// TIA Portal V20 export
FUNCTION_BLOCK "LER_Vision_XGX2000_Conversion"   // FB157, LAD
// stored: Access Published, MemoryReserve 100, SetENOAutomatically false
   VAR_INPUT
      VisionData : "LER_typeVisionMonitoring";
   END_VAR
   VAR_OUTPUT
      VisionDataConvert : "LER_typeVisionResultData";
   END_VAR
BEGIN

REGION Network 1: Stack_Width_Judgement Result (0:NONE,1:OK,2:NG)
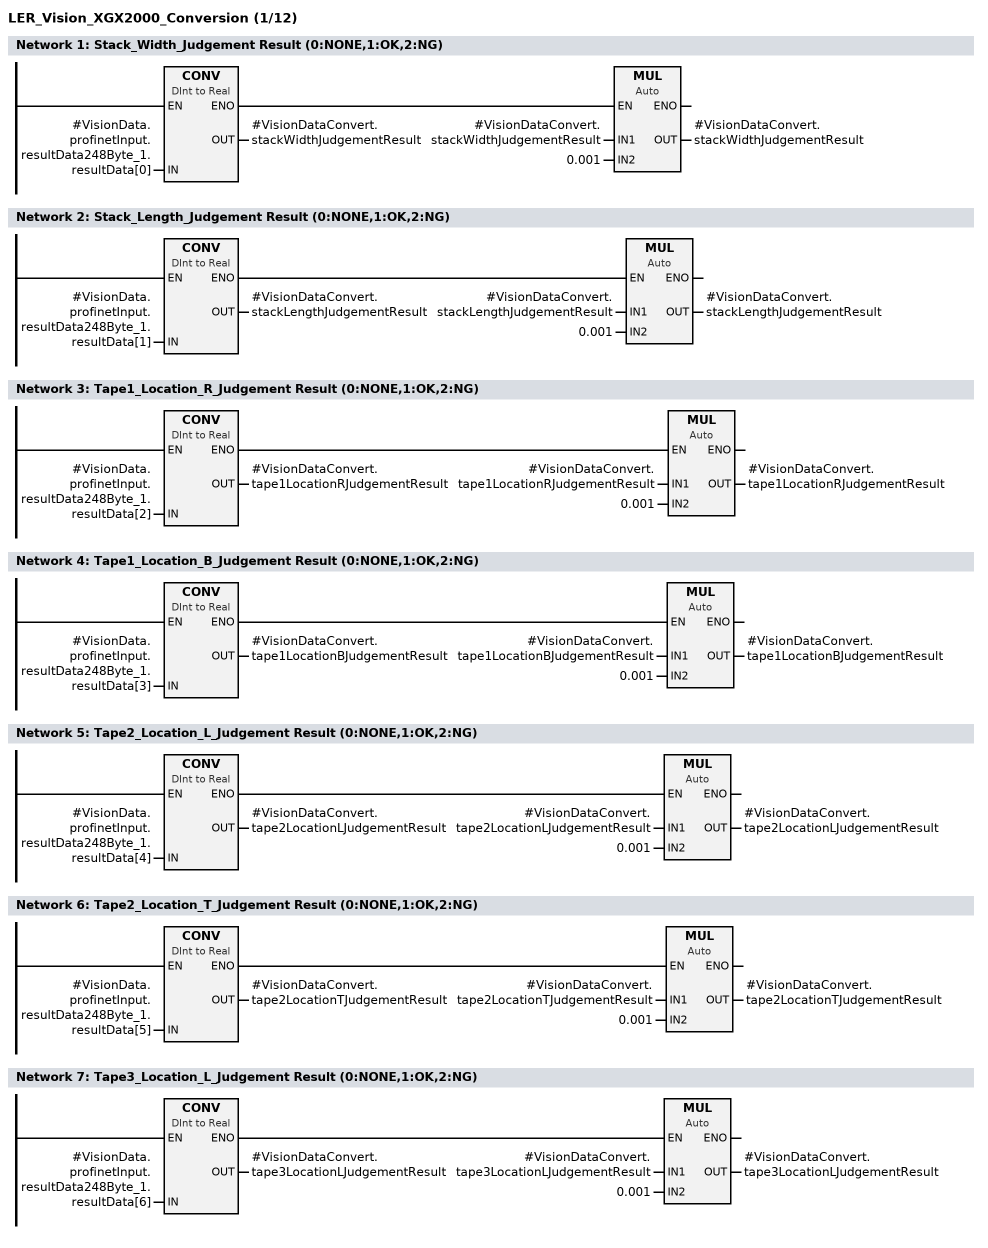
   RUNG wire#powerrail
      { S7_Templates := "[SrcType := DInt, DestType := Real]" } Convert(in := #VisionData.profinetInput.resultData248Byte_1.resultData[0], out => #VisionDataConvert.stackWidthJudgementResult)
      Mul(in1 := #VisionDataConvert.stackWidthJudgementResult, in2 := 0.001, out => #VisionDataConvert.stackWidthJudgementResult)
   END_RUNG
   // the same network as SCL:
   #VisionDataConvert.stackWidthJudgementResult := DINT_TO_REAL(#VisionData.profinetInput.resultData248Byte_1.resultData[0]);
   #VisionDataConvert.stackWidthJudgementResult := #VisionDataConvert.stackWidthJudgementResult * 0.001;
END_REGION

REGION Network 2: Stack_Length_Judgement Result (0:NONE,1:OK,2:NG)
   RUNG wire#powerrail
      { S7_Templates := "[SrcType := DInt, DestType := Real]" } Convert(in := #VisionData.profinetInput.resultData248Byte_1.resultData[1], out => #VisionDataConvert.stackLengthJudgementResult)
      Mul(in1 := #VisionDataConvert.stackLengthJudgementResult, in2 := 0.001, out => #VisionDataConvert.stackLengthJudgementResult)
   END_RUNG
   // the same network as SCL:
   #VisionDataConvert.stackLengthJudgementResult := DINT_TO_REAL(#VisionData.profinetInput.resultData248Byte_1.resultData[1]);
   #VisionDataConvert.stackLengthJudgementResult := #VisionDataConvert.stackLengthJudgementResult * 0.001;
END_REGION

REGION Network 3: Tape1_Location_R_Judgement Result (0:NONE,1:OK,2:NG)
   RUNG wire#powerrail
      { S7_Templates := "[SrcType := DInt, DestType := Real]" } Convert(in := #VisionData.profinetInput.resultData248Byte_1.resultData[2], out => #VisionDataConvert.tape1LocationRJudgementResult)
      Mul(in1 := #VisionDataConvert.tape1LocationRJudgementResult, in2 := 0.001, out => #VisionDataConvert.tape1LocationRJudgementResult)
   END_RUNG
   // the same network as SCL:
   #VisionDataConvert.tape1LocationRJudgementResult := DINT_TO_REAL(#VisionData.profinetInput.resultData248Byte_1.resultData[2]);
   #VisionDataConvert.tape1LocationRJudgementResult := #VisionDataConvert.tape1LocationRJudgementResult * 0.001;
END_REGION

REGION Network 4: Tape1_Location_B_Judgement Result (0:NONE,1:OK,2:NG)
   RUNG wire#powerrail
      { S7_Templates := "[SrcType := DInt, DestType := Real]" } Convert(in := #VisionData.profinetInput.resultData248Byte_1.resultData[3], out => #VisionDataConvert.tape1LocationBJudgementResult)
      Mul(in1 := #VisionDataConvert.tape1LocationBJudgementResult, in2 := 0.001, out => #VisionDataConvert.tape1LocationBJudgementResult)
   END_RUNG
   // the same network as SCL:
   #VisionDataConvert.tape1LocationBJudgementResult := DINT_TO_REAL(#VisionData.profinetInput.resultData248Byte_1.resultData[3]);
   #VisionDataConvert.tape1LocationBJudgementResult := #VisionDataConvert.tape1LocationBJudgementResult * 0.001;
END_REGION

REGION Network 5: Tape2_Location_L_Judgement Result (0:NONE,1:OK,2:NG)
   RUNG wire#powerrail
      { S7_Templates := "[SrcType := DInt, DestType := Real]" } Convert(in := #VisionData.profinetInput.resultData248Byte_1.resultData[4], out => #VisionDataConvert.tape2LocationLJudgementResult)
      Mul(in1 := #VisionDataConvert.tape2LocationLJudgementResult, in2 := 0.001, out => #VisionDataConvert.tape2LocationLJudgementResult)
   END_RUNG
   // the same network as SCL:
   #VisionDataConvert.tape2LocationLJudgementResult := DINT_TO_REAL(#VisionData.profinetInput.resultData248Byte_1.resultData[4]);
   #VisionDataConvert.tape2LocationLJudgementResult := #VisionDataConvert.tape2LocationLJudgementResult * 0.001;
END_REGION

REGION Network 6: Tape2_Location_T_Judgement Result (0:NONE,1:OK,2:NG)
   RUNG wire#powerrail
      { S7_Templates := "[SrcType := DInt, DestType := Real]" } Convert(in := #VisionData.profinetInput.resultData248Byte_1.resultData[5], out => #VisionDataConvert.tape2LocationTJudgementResult)
      Mul(in1 := #VisionDataConvert.tape2LocationTJudgementResult, in2 := 0.001, out => #VisionDataConvert.tape2LocationTJudgementResult)
   END_RUNG
   // the same network as SCL:
   #VisionDataConvert.tape2LocationTJudgementResult := DINT_TO_REAL(#VisionData.profinetInput.resultData248Byte_1.resultData[5]);
   #VisionDataConvert.tape2LocationTJudgementResult := #VisionDataConvert.tape2LocationTJudgementResult * 0.001;
END_REGION

REGION Network 7: Tape3_Location_L_Judgement Result (0:NONE,1:OK,2:NG)
   RUNG wire#powerrail
      { S7_Templates := "[SrcType := DInt, DestType := Real]" } Convert(in := #VisionData.profinetInput.resultData248Byte_1.resultData[6], out => #VisionDataConvert.tape3LocationLJudgementResult)
      Mul(in1 := #VisionDataConvert.tape3LocationLJudgementResult, in2 := 0.001, out => #VisionDataConvert.tape3LocationLJudgementResult)
   END_RUNG
   // the same network as SCL:
   #VisionDataConvert.tape3LocationLJudgementResult := DINT_TO_REAL(#VisionData.profinetInput.resultData248Byte_1.resultData[6]);
   #VisionDataConvert.tape3LocationLJudgementResult := #VisionDataConvert.tape3LocationLJudgementResult * 0.001;
END_REGION

REGION Network 8: Tape3_Location_B_Judgement Result (0:NONE,1:OK,2:NG)
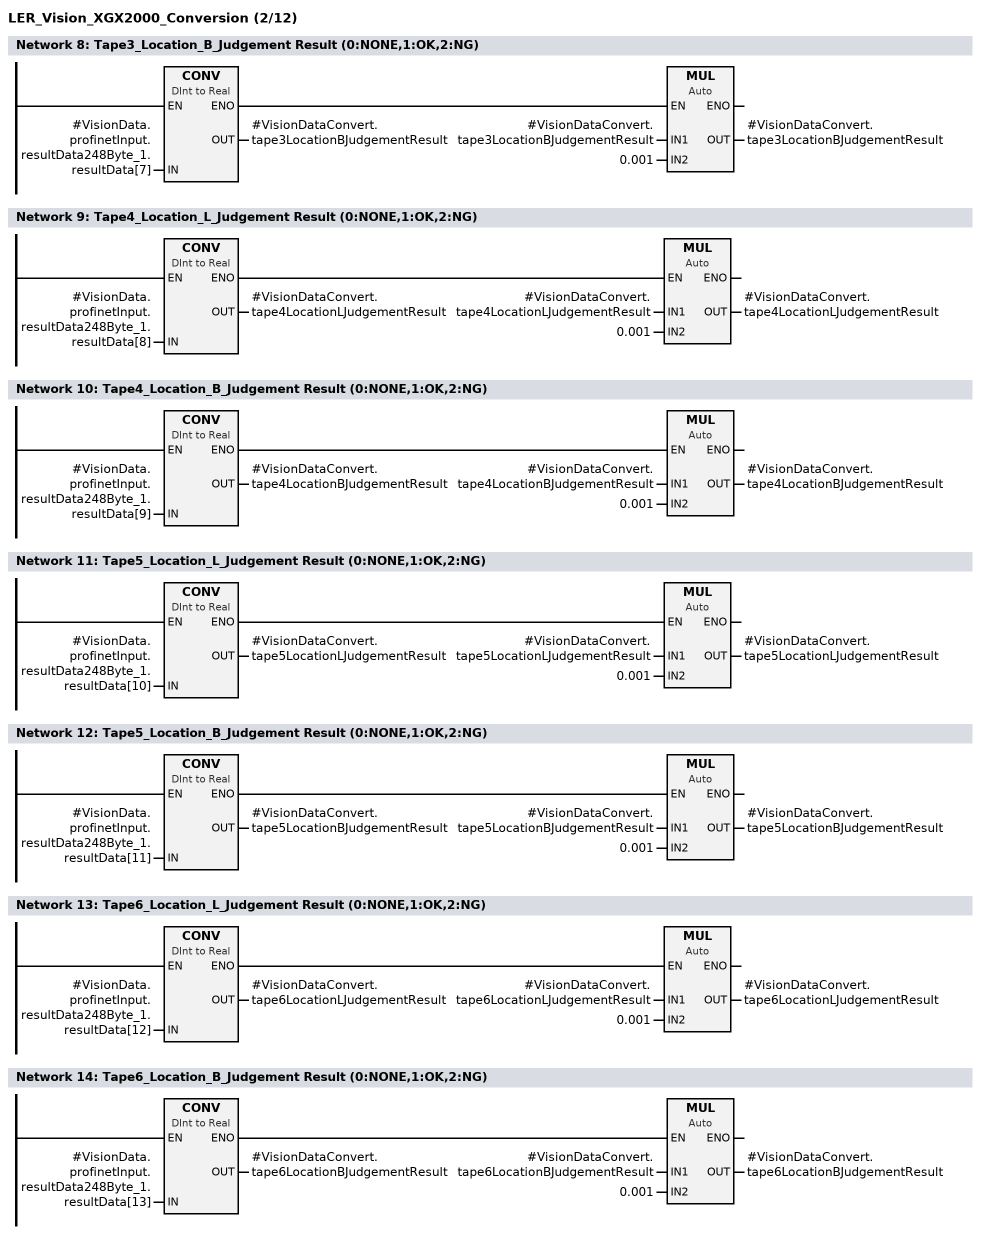
   RUNG wire#powerrail
      { S7_Templates := "[SrcType := DInt, DestType := Real]" } Convert(in := #VisionData.profinetInput.resultData248Byte_1.resultData[7], out => #VisionDataConvert.tape3LocationBJudgementResult)
      Mul(in1 := #VisionDataConvert.tape3LocationBJudgementResult, in2 := 0.001, out => #VisionDataConvert.tape3LocationBJudgementResult)
   END_RUNG
   // the same network as SCL:
   #VisionDataConvert.tape3LocationBJudgementResult := DINT_TO_REAL(#VisionData.profinetInput.resultData248Byte_1.resultData[7]);
   #VisionDataConvert.tape3LocationBJudgementResult := #VisionDataConvert.tape3LocationBJudgementResult * 0.001;
END_REGION

REGION Network 9: Tape4_Location_L_Judgement Result (0:NONE,1:OK,2:NG)
   RUNG wire#powerrail
      { S7_Templates := "[SrcType := DInt, DestType := Real]" } Convert(in := #VisionData.profinetInput.resultData248Byte_1.resultData[8], out => #VisionDataConvert.tape4LocationLJudgementResult)
      Mul(in1 := #VisionDataConvert.tape4LocationLJudgementResult, in2 := 0.001, out => #VisionDataConvert.tape4LocationLJudgementResult)
   END_RUNG
   // the same network as SCL:
   #VisionDataConvert.tape4LocationLJudgementResult := DINT_TO_REAL(#VisionData.profinetInput.resultData248Byte_1.resultData[8]);
   #VisionDataConvert.tape4LocationLJudgementResult := #VisionDataConvert.tape4LocationLJudgementResult * 0.001;
END_REGION

REGION Network 10: Tape4_Location_B_Judgement Result (0:NONE,1:OK,2:NG)
   RUNG wire#powerrail
      { S7_Templates := "[SrcType := DInt, DestType := Real]" } Convert(in := #VisionData.profinetInput.resultData248Byte_1.resultData[9], out => #VisionDataConvert.tape4LocationBJudgementResult)
      Mul(in1 := #VisionDataConvert.tape4LocationBJudgementResult, in2 := 0.001, out => #VisionDataConvert.tape4LocationBJudgementResult)
   END_RUNG
   // the same network as SCL:
   #VisionDataConvert.tape4LocationBJudgementResult := DINT_TO_REAL(#VisionData.profinetInput.resultData248Byte_1.resultData[9]);
   #VisionDataConvert.tape4LocationBJudgementResult := #VisionDataConvert.tape4LocationBJudgementResult * 0.001;
END_REGION

REGION Network 11: Tape5_Location_L_Judgement Result (0:NONE,1:OK,2:NG)
   RUNG wire#powerrail
      { S7_Templates := "[SrcType := DInt, DestType := Real]" } Convert(in := #VisionData.profinetInput.resultData248Byte_1.resultData[10], out => #VisionDataConvert.tape5LocationLJudgementResult)
      Mul(in1 := #VisionDataConvert.tape5LocationLJudgementResult, in2 := 0.001, out => #VisionDataConvert.tape5LocationLJudgementResult)
   END_RUNG
   // the same network as SCL:
   #VisionDataConvert.tape5LocationLJudgementResult := DINT_TO_REAL(#VisionData.profinetInput.resultData248Byte_1.resultData[10]);
   #VisionDataConvert.tape5LocationLJudgementResult := #VisionDataConvert.tape5LocationLJudgementResult * 0.001;
END_REGION

REGION Network 12: Tape5_Location_B_Judgement Result (0:NONE,1:OK,2:NG)
   RUNG wire#powerrail
      { S7_Templates := "[SrcType := DInt, DestType := Real]" } Convert(in := #VisionData.profinetInput.resultData248Byte_1.resultData[11], out => #VisionDataConvert.tape5LocationBJudgementResult)
      Mul(in1 := #VisionDataConvert.tape5LocationBJudgementResult, in2 := 0.001, out => #VisionDataConvert.tape5LocationBJudgementResult)
   END_RUNG
   // the same network as SCL:
   #VisionDataConvert.tape5LocationBJudgementResult := DINT_TO_REAL(#VisionData.profinetInput.resultData248Byte_1.resultData[11]);
   #VisionDataConvert.tape5LocationBJudgementResult := #VisionDataConvert.tape5LocationBJudgementResult * 0.001;
END_REGION

REGION Network 13: Tape6_Location_L_Judgement Result (0:NONE,1:OK,2:NG)
   RUNG wire#powerrail
      { S7_Templates := "[SrcType := DInt, DestType := Real]" } Convert(in := #VisionData.profinetInput.resultData248Byte_1.resultData[12], out => #VisionDataConvert.tape6LocationLJudgementResult)
      Mul(in1 := #VisionDataConvert.tape6LocationLJudgementResult, in2 := 0.001, out => #VisionDataConvert.tape6LocationLJudgementResult)
   END_RUNG
   // the same network as SCL:
   #VisionDataConvert.tape6LocationLJudgementResult := DINT_TO_REAL(#VisionData.profinetInput.resultData248Byte_1.resultData[12]);
   #VisionDataConvert.tape6LocationLJudgementResult := #VisionDataConvert.tape6LocationLJudgementResult * 0.001;
END_REGION

REGION Network 14: Tape6_Location_B_Judgement Result (0:NONE,1:OK,2:NG)
   RUNG wire#powerrail
      { S7_Templates := "[SrcType := DInt, DestType := Real]" } Convert(in := #VisionData.profinetInput.resultData248Byte_1.resultData[13], out => #VisionDataConvert.tape6LocationBJudgementResult)
      Mul(in1 := #VisionDataConvert.tape6LocationBJudgementResult, in2 := 0.001, out => #VisionDataConvert.tape6LocationBJudgementResult)
   END_RUNG
   // the same network as SCL:
   #VisionDataConvert.tape6LocationBJudgementResult := DINT_TO_REAL(#VisionData.profinetInput.resultData248Byte_1.resultData[13]);
   #VisionDataConvert.tape6LocationBJudgementResult := #VisionDataConvert.tape6LocationBJudgementResult * 0.001;
END_REGION

REGION Network 15: Tape7_Location_L_Judgement Result (0:NONE,1:OK,2:NG)
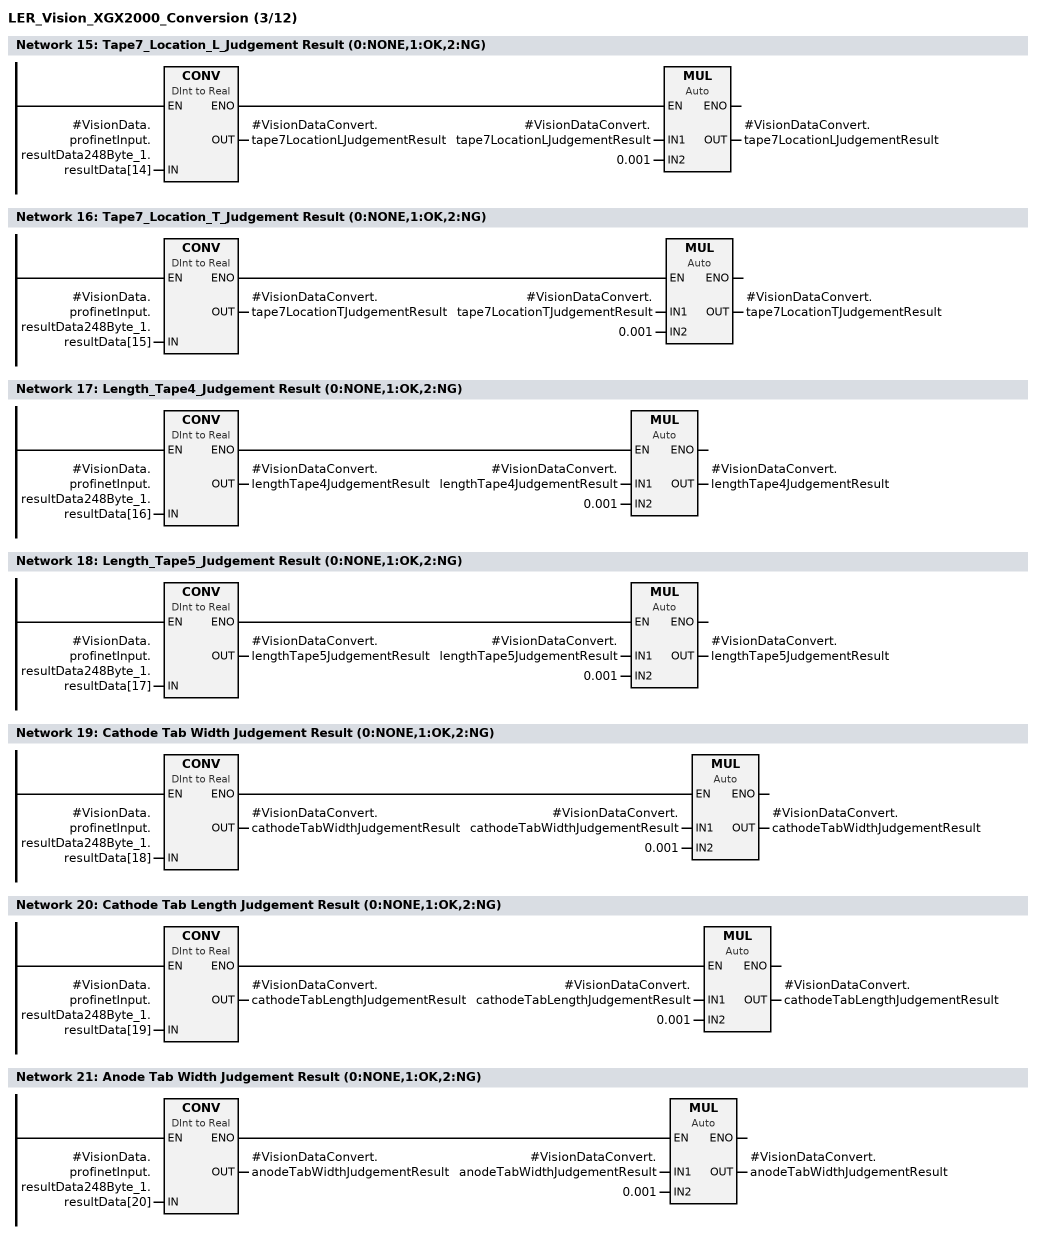
   RUNG wire#powerrail
      { S7_Templates := "[SrcType := DInt, DestType := Real]" } Convert(in := #VisionData.profinetInput.resultData248Byte_1.resultData[14], out => #VisionDataConvert.tape7LocationLJudgementResult)
      Mul(in1 := #VisionDataConvert.tape7LocationLJudgementResult, in2 := 0.001, out => #VisionDataConvert.tape7LocationLJudgementResult)
   END_RUNG
   // the same network as SCL:
   #VisionDataConvert.tape7LocationLJudgementResult := DINT_TO_REAL(#VisionData.profinetInput.resultData248Byte_1.resultData[14]);
   #VisionDataConvert.tape7LocationLJudgementResult := #VisionDataConvert.tape7LocationLJudgementResult * 0.001;
END_REGION

REGION Network 16: Tape7_Location_T_Judgement Result (0:NONE,1:OK,2:NG)
   RUNG wire#powerrail
      { S7_Templates := "[SrcType := DInt, DestType := Real]" } Convert(in := #VisionData.profinetInput.resultData248Byte_1.resultData[15], out => #VisionDataConvert.tape7LocationTJudgementResult)
      Mul(in1 := #VisionDataConvert.tape7LocationTJudgementResult, in2 := 0.001, out => #VisionDataConvert.tape7LocationTJudgementResult)
   END_RUNG
   // the same network as SCL:
   #VisionDataConvert.tape7LocationTJudgementResult := DINT_TO_REAL(#VisionData.profinetInput.resultData248Byte_1.resultData[15]);
   #VisionDataConvert.tape7LocationTJudgementResult := #VisionDataConvert.tape7LocationTJudgementResult * 0.001;
END_REGION

REGION Network 17: Length_Tape4_Judgement Result (0:NONE,1:OK,2:NG)
   RUNG wire#powerrail
      { S7_Templates := "[SrcType := DInt, DestType := Real]" } Convert(in := #VisionData.profinetInput.resultData248Byte_1.resultData[16], out => #VisionDataConvert.lengthTape4JudgementResult)
      Mul(in1 := #VisionDataConvert.lengthTape4JudgementResult, in2 := 0.001, out => #VisionDataConvert.lengthTape4JudgementResult)
   END_RUNG
   // the same network as SCL:
   #VisionDataConvert.lengthTape4JudgementResult := DINT_TO_REAL(#VisionData.profinetInput.resultData248Byte_1.resultData[16]);
   #VisionDataConvert.lengthTape4JudgementResult := #VisionDataConvert.lengthTape4JudgementResult * 0.001;
END_REGION

REGION Network 18: Length_Tape5_Judgement Result (0:NONE,1:OK,2:NG)
   RUNG wire#powerrail
      { S7_Templates := "[SrcType := DInt, DestType := Real]" } Convert(in := #VisionData.profinetInput.resultData248Byte_1.resultData[17], out => #VisionDataConvert.lengthTape5JudgementResult)
      Mul(in1 := #VisionDataConvert.lengthTape5JudgementResult, in2 := 0.001, out => #VisionDataConvert.lengthTape5JudgementResult)
   END_RUNG
   // the same network as SCL:
   #VisionDataConvert.lengthTape5JudgementResult := DINT_TO_REAL(#VisionData.profinetInput.resultData248Byte_1.resultData[17]);
   #VisionDataConvert.lengthTape5JudgementResult := #VisionDataConvert.lengthTape5JudgementResult * 0.001;
END_REGION

REGION Network 19: Cathode Tab Width Judgement Result (0:NONE,1:OK,2:NG)
   RUNG wire#powerrail
      { S7_Templates := "[SrcType := DInt, DestType := Real]" } Convert(in := #VisionData.profinetInput.resultData248Byte_1.resultData[18], out => #VisionDataConvert.cathodeTabWidthJudgementResult)
      Mul(in1 := #VisionDataConvert.cathodeTabWidthJudgementResult, in2 := 0.001, out => #VisionDataConvert.cathodeTabWidthJudgementResult)
   END_RUNG
   // the same network as SCL:
   #VisionDataConvert.cathodeTabWidthJudgementResult := DINT_TO_REAL(#VisionData.profinetInput.resultData248Byte_1.resultData[18]);
   #VisionDataConvert.cathodeTabWidthJudgementResult := #VisionDataConvert.cathodeTabWidthJudgementResult * 0.001;
END_REGION

REGION Network 20: Cathode Tab Length Judgement Result (0:NONE,1:OK,2:NG)
   RUNG wire#powerrail
      { S7_Templates := "[SrcType := DInt, DestType := Real]" } Convert(in := #VisionData.profinetInput.resultData248Byte_1.resultData[19], out => #VisionDataConvert.cathodeTabLengthJudgementResult)
      Mul(in1 := #VisionDataConvert.cathodeTabLengthJudgementResult, in2 := 0.001, out => #VisionDataConvert.cathodeTabLengthJudgementResult)
   END_RUNG
   // the same network as SCL:
   #VisionDataConvert.cathodeTabLengthJudgementResult := DINT_TO_REAL(#VisionData.profinetInput.resultData248Byte_1.resultData[19]);
   #VisionDataConvert.cathodeTabLengthJudgementResult := #VisionDataConvert.cathodeTabLengthJudgementResult * 0.001;
END_REGION

REGION Network 21: Anode Tab Width Judgement Result (0:NONE,1:OK,2:NG)
   RUNG wire#powerrail
      { S7_Templates := "[SrcType := DInt, DestType := Real]" } Convert(in := #VisionData.profinetInput.resultData248Byte_1.resultData[20], out => #VisionDataConvert.anodeTabWidthJudgementResult)
      Mul(in1 := #VisionDataConvert.anodeTabWidthJudgementResult, in2 := 0.001, out => #VisionDataConvert.anodeTabWidthJudgementResult)
   END_RUNG
   // the same network as SCL:
   #VisionDataConvert.anodeTabWidthJudgementResult := DINT_TO_REAL(#VisionData.profinetInput.resultData248Byte_1.resultData[20]);
   #VisionDataConvert.anodeTabWidthJudgementResult := #VisionDataConvert.anodeTabWidthJudgementResult * 0.001;
END_REGION

REGION Network 22: Anode Tab Length Judgement Result (0:NONE,1:OK,2:NG)
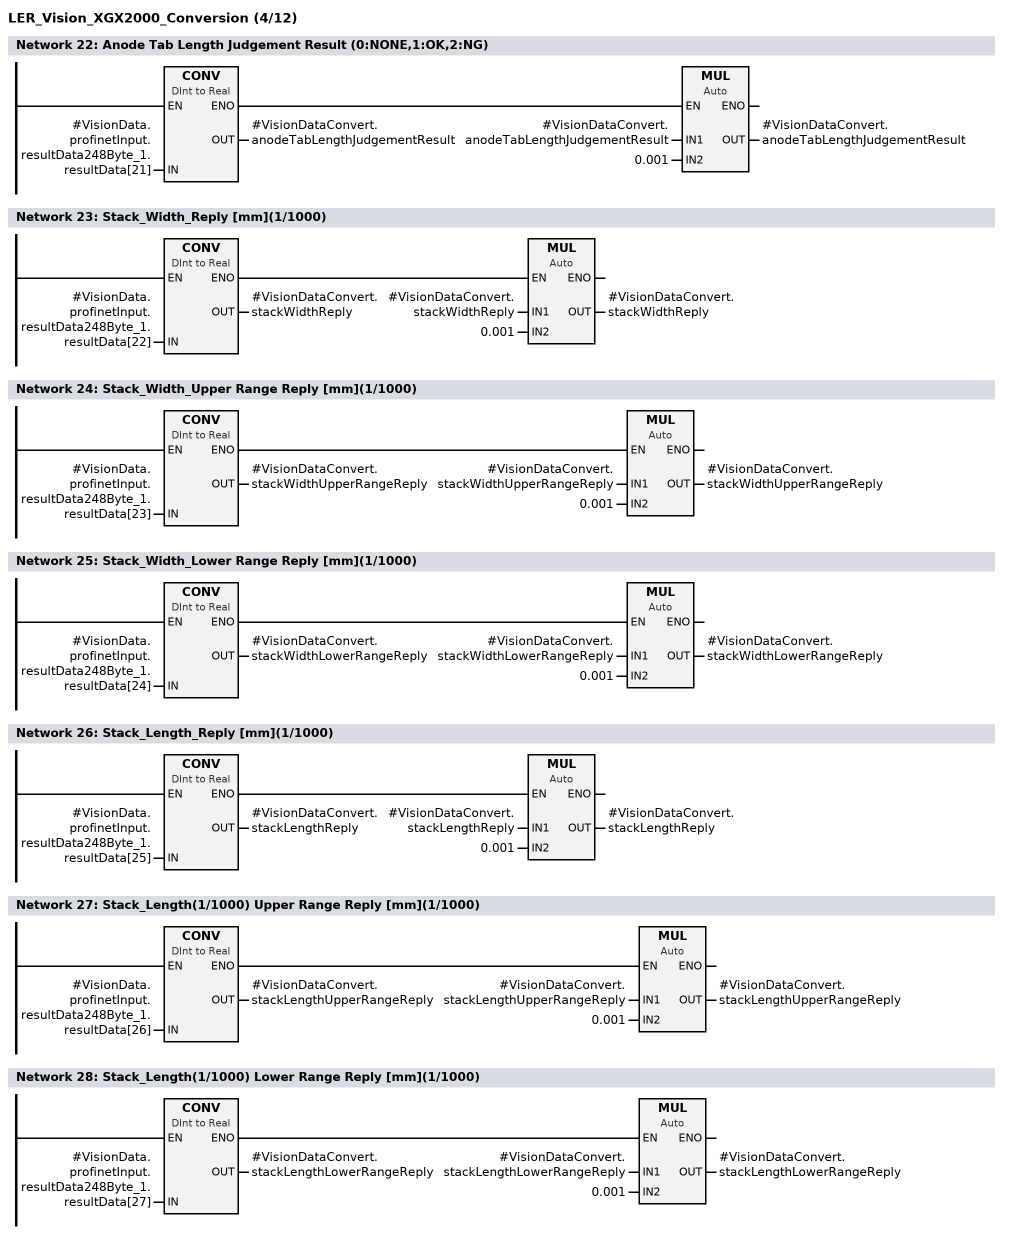
   RUNG wire#powerrail
      { S7_Templates := "[SrcType := DInt, DestType := Real]" } Convert(in := #VisionData.profinetInput.resultData248Byte_1.resultData[21], out => #VisionDataConvert.anodeTabLengthJudgementResult)
      Mul(in1 := #VisionDataConvert.anodeTabLengthJudgementResult, in2 := 0.001, out => #VisionDataConvert.anodeTabLengthJudgementResult)
   END_RUNG
   // the same network as SCL:
   #VisionDataConvert.anodeTabLengthJudgementResult := DINT_TO_REAL(#VisionData.profinetInput.resultData248Byte_1.resultData[21]);
   #VisionDataConvert.anodeTabLengthJudgementResult := #VisionDataConvert.anodeTabLengthJudgementResult * 0.001;
END_REGION

REGION Network 23: Stack_Width_Reply [mm](1/1000)
   RUNG wire#powerrail
      { S7_Templates := "[SrcType := DInt, DestType := Real]" } Convert(in := #VisionData.profinetInput.resultData248Byte_1.resultData[22], out => #VisionDataConvert.stackWidthReply)
      Mul(in1 := #VisionDataConvert.stackWidthReply, in2 := 0.001, out => #VisionDataConvert.stackWidthReply)
   END_RUNG
   // the same network as SCL:
   #VisionDataConvert.stackWidthReply := DINT_TO_REAL(#VisionData.profinetInput.resultData248Byte_1.resultData[22]);
   #VisionDataConvert.stackWidthReply := #VisionDataConvert.stackWidthReply * 0.001;
END_REGION

REGION Network 24: Stack_Width_Upper Range Reply [mm](1/1000)
   RUNG wire#powerrail
      { S7_Templates := "[SrcType := DInt, DestType := Real]" } Convert(in := #VisionData.profinetInput.resultData248Byte_1.resultData[23], out => #VisionDataConvert.stackWidthUpperRangeReply)
      Mul(in1 := #VisionDataConvert.stackWidthUpperRangeReply, in2 := 0.001, out => #VisionDataConvert.stackWidthUpperRangeReply)
   END_RUNG
   // the same network as SCL:
   #VisionDataConvert.stackWidthUpperRangeReply := DINT_TO_REAL(#VisionData.profinetInput.resultData248Byte_1.resultData[23]);
   #VisionDataConvert.stackWidthUpperRangeReply := #VisionDataConvert.stackWidthUpperRangeReply * 0.001;
END_REGION

REGION Network 25: Stack_Width_Lower Range Reply [mm](1/1000)
   RUNG wire#powerrail
      { S7_Templates := "[SrcType := DInt, DestType := Real]" } Convert(in := #VisionData.profinetInput.resultData248Byte_1.resultData[24], out => #VisionDataConvert.stackWidthLowerRangeReply)
      Mul(in1 := #VisionDataConvert.stackWidthLowerRangeReply, in2 := 0.001, out => #VisionDataConvert.stackWidthLowerRangeReply)
   END_RUNG
   // the same network as SCL:
   #VisionDataConvert.stackWidthLowerRangeReply := DINT_TO_REAL(#VisionData.profinetInput.resultData248Byte_1.resultData[24]);
   #VisionDataConvert.stackWidthLowerRangeReply := #VisionDataConvert.stackWidthLowerRangeReply * 0.001;
END_REGION

REGION Network 26: Stack_Length_Reply [mm](1/1000)
   RUNG wire#powerrail
      { S7_Templates := "[SrcType := DInt, DestType := Real]" } Convert(in := #VisionData.profinetInput.resultData248Byte_1.resultData[25], out => #VisionDataConvert.stackLengthReply)
      Mul(in1 := #VisionDataConvert.stackLengthReply, in2 := 0.001, out => #VisionDataConvert.stackLengthReply)
   END_RUNG
   // the same network as SCL:
   #VisionDataConvert.stackLengthReply := DINT_TO_REAL(#VisionData.profinetInput.resultData248Byte_1.resultData[25]);
   #VisionDataConvert.stackLengthReply := #VisionDataConvert.stackLengthReply * 0.001;
END_REGION

REGION Network 27: Stack_Length(1/1000) Upper Range Reply [mm](1/1000)
   RUNG wire#powerrail
      { S7_Templates := "[SrcType := DInt, DestType := Real]" } Convert(in := #VisionData.profinetInput.resultData248Byte_1.resultData[26], out => #VisionDataConvert.stackLengthUpperRangeReply)
      Mul(in1 := #VisionDataConvert.stackLengthUpperRangeReply, in2 := 0.001, out => #VisionDataConvert.stackLengthUpperRangeReply)
   END_RUNG
   // the same network as SCL:
   #VisionDataConvert.stackLengthUpperRangeReply := DINT_TO_REAL(#VisionData.profinetInput.resultData248Byte_1.resultData[26]);
   #VisionDataConvert.stackLengthUpperRangeReply := #VisionDataConvert.stackLengthUpperRangeReply * 0.001;
END_REGION

REGION Network 28: Stack_Length(1/1000) Lower Range Reply [mm](1/1000)
   RUNG wire#powerrail
      { S7_Templates := "[SrcType := DInt, DestType := Real]" } Convert(in := #VisionData.profinetInput.resultData248Byte_1.resultData[27], out => #VisionDataConvert.stackLengthLowerRangeReply)
      Mul(in1 := #VisionDataConvert.stackLengthLowerRangeReply, in2 := 0.001, out => #VisionDataConvert.stackLengthLowerRangeReply)
   END_RUNG
   // the same network as SCL:
   #VisionDataConvert.stackLengthLowerRangeReply := DINT_TO_REAL(#VisionData.profinetInput.resultData248Byte_1.resultData[27]);
   #VisionDataConvert.stackLengthLowerRangeReply := #VisionDataConvert.stackLengthLowerRangeReply * 0.001;
END_REGION

REGION Network 29: Tape1_Location_R_Reply [mm](1/1000)
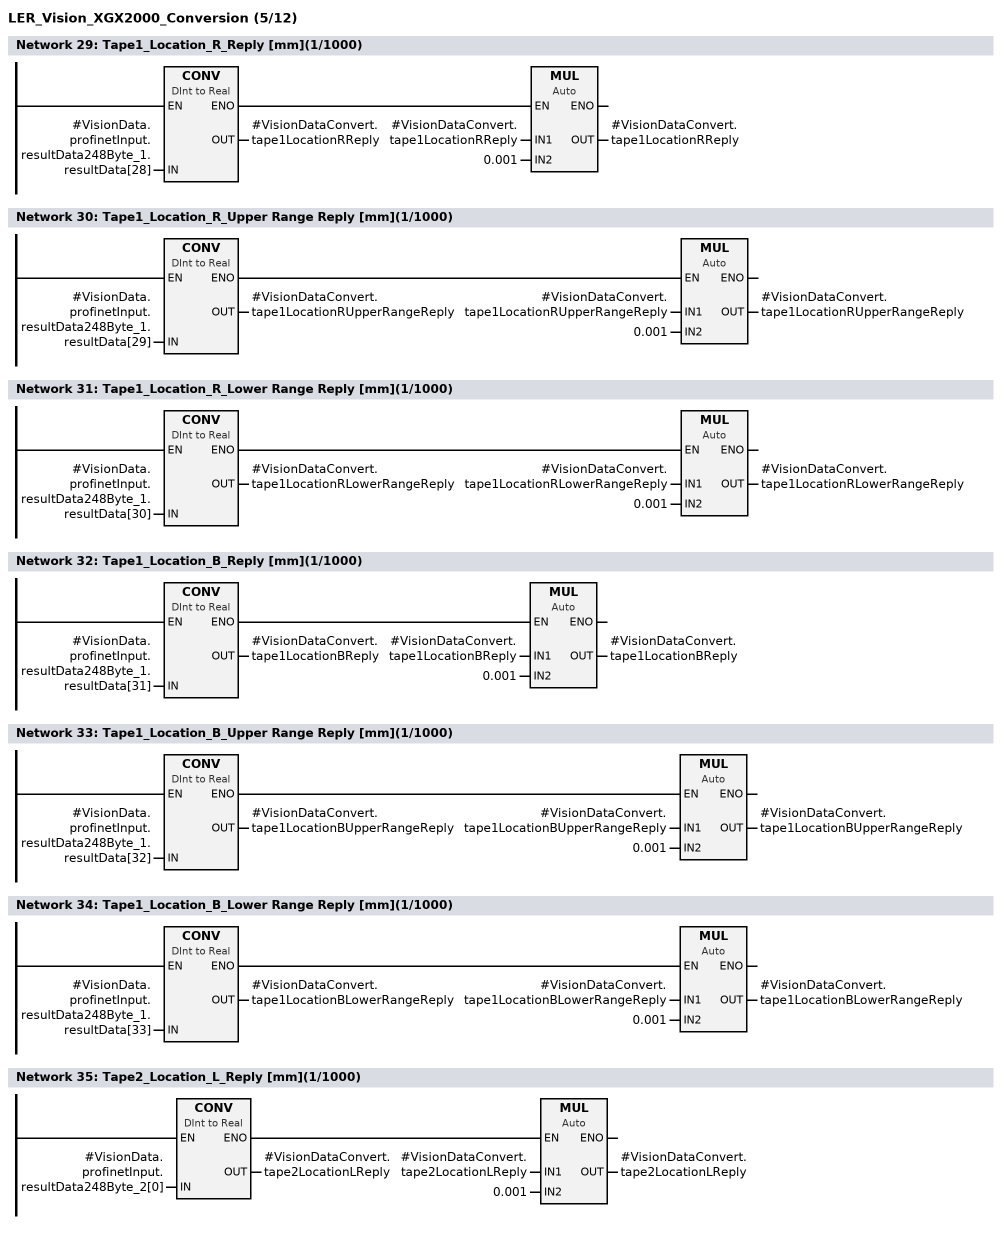
   RUNG wire#powerrail
      { S7_Templates := "[SrcType := DInt, DestType := Real]" } Convert(in := #VisionData.profinetInput.resultData248Byte_1.resultData[28], out => #VisionDataConvert.tape1LocationRReply)
      Mul(in1 := #VisionDataConvert.tape1LocationRReply, in2 := 0.001, out => #VisionDataConvert.tape1LocationRReply)
   END_RUNG
   // the same network as SCL:
   #VisionDataConvert.tape1LocationRReply := DINT_TO_REAL(#VisionData.profinetInput.resultData248Byte_1.resultData[28]);
   #VisionDataConvert.tape1LocationRReply := #VisionDataConvert.tape1LocationRReply * 0.001;
END_REGION

REGION Network 30: Tape1_Location_R_Upper Range Reply [mm](1/1000)
   RUNG wire#powerrail
      { S7_Templates := "[SrcType := DInt, DestType := Real]" } Convert(in := #VisionData.profinetInput.resultData248Byte_1.resultData[29], out => #VisionDataConvert.tape1LocationRUpperRangeReply)
      Mul(in1 := #VisionDataConvert.tape1LocationRUpperRangeReply, in2 := 0.001, out => #VisionDataConvert.tape1LocationRUpperRangeReply)
   END_RUNG
   // the same network as SCL:
   #VisionDataConvert.tape1LocationRUpperRangeReply := DINT_TO_REAL(#VisionData.profinetInput.resultData248Byte_1.resultData[29]);
   #VisionDataConvert.tape1LocationRUpperRangeReply := #VisionDataConvert.tape1LocationRUpperRangeReply * 0.001;
END_REGION

REGION Network 31: Tape1_Location_R_Lower Range Reply [mm](1/1000)
   RUNG wire#powerrail
      { S7_Templates := "[SrcType := DInt, DestType := Real]" } Convert(in := #VisionData.profinetInput.resultData248Byte_1.resultData[30], out => #VisionDataConvert.tape1LocationRLowerRangeReply)
      Mul(in1 := #VisionDataConvert.tape1LocationRLowerRangeReply, in2 := 0.001, out => #VisionDataConvert.tape1LocationRLowerRangeReply)
   END_RUNG
   // the same network as SCL:
   #VisionDataConvert.tape1LocationRLowerRangeReply := DINT_TO_REAL(#VisionData.profinetInput.resultData248Byte_1.resultData[30]);
   #VisionDataConvert.tape1LocationRLowerRangeReply := #VisionDataConvert.tape1LocationRLowerRangeReply * 0.001;
END_REGION

REGION Network 32: Tape1_Location_B_Reply [mm](1/1000)
   RUNG wire#powerrail
      { S7_Templates := "[SrcType := DInt, DestType := Real]" } Convert(in := #VisionData.profinetInput.resultData248Byte_1.resultData[31], out => #VisionDataConvert.tape1LocationBReply)
      Mul(in1 := #VisionDataConvert.tape1LocationBReply, in2 := 0.001, out => #VisionDataConvert.tape1LocationBReply)
   END_RUNG
   // the same network as SCL:
   #VisionDataConvert.tape1LocationBReply := DINT_TO_REAL(#VisionData.profinetInput.resultData248Byte_1.resultData[31]);
   #VisionDataConvert.tape1LocationBReply := #VisionDataConvert.tape1LocationBReply * 0.001;
END_REGION

REGION Network 33: Tape1_Location_B_Upper Range Reply [mm](1/1000)
   RUNG wire#powerrail
      { S7_Templates := "[SrcType := DInt, DestType := Real]" } Convert(in := #VisionData.profinetInput.resultData248Byte_1.resultData[32], out => #VisionDataConvert.tape1LocationBUpperRangeReply)
      Mul(in1 := #VisionDataConvert.tape1LocationBUpperRangeReply, in2 := 0.001, out => #VisionDataConvert.tape1LocationBUpperRangeReply)
   END_RUNG
   // the same network as SCL:
   #VisionDataConvert.tape1LocationBUpperRangeReply := DINT_TO_REAL(#VisionData.profinetInput.resultData248Byte_1.resultData[32]);
   #VisionDataConvert.tape1LocationBUpperRangeReply := #VisionDataConvert.tape1LocationBUpperRangeReply * 0.001;
END_REGION

REGION Network 34: Tape1_Location_B_Lower Range Reply [mm](1/1000)
   RUNG wire#powerrail
      { S7_Templates := "[SrcType := DInt, DestType := Real]" } Convert(in := #VisionData.profinetInput.resultData248Byte_1.resultData[33], out => #VisionDataConvert.tape1LocationBLowerRangeReply)
      Mul(in1 := #VisionDataConvert.tape1LocationBLowerRangeReply, in2 := 0.001, out => #VisionDataConvert.tape1LocationBLowerRangeReply)
   END_RUNG
   // the same network as SCL:
   #VisionDataConvert.tape1LocationBLowerRangeReply := DINT_TO_REAL(#VisionData.profinetInput.resultData248Byte_1.resultData[33]);
   #VisionDataConvert.tape1LocationBLowerRangeReply := #VisionDataConvert.tape1LocationBLowerRangeReply * 0.001;
END_REGION

REGION Network 35: Tape2_Location_L_Reply [mm](1/1000)
   RUNG wire#powerrail
      { S7_Templates := "[SrcType := DInt, DestType := Real]" } Convert(in := #VisionData.profinetInput.resultData248Byte_2[0], out => #VisionDataConvert.tape2LocationLReply)
      Mul(in1 := #VisionDataConvert.tape2LocationLReply, in2 := 0.001, out => #VisionDataConvert.tape2LocationLReply)
   END_RUNG
   // the same network as SCL:
   #VisionDataConvert.tape2LocationLReply := DINT_TO_REAL(#VisionData.profinetInput.resultData248Byte_2[0]);
   #VisionDataConvert.tape2LocationLReply := #VisionDataConvert.tape2LocationLReply * 0.001;
END_REGION

REGION Network 36: Tape2_Location_L_Upper Range Reply [mm](1/1000)
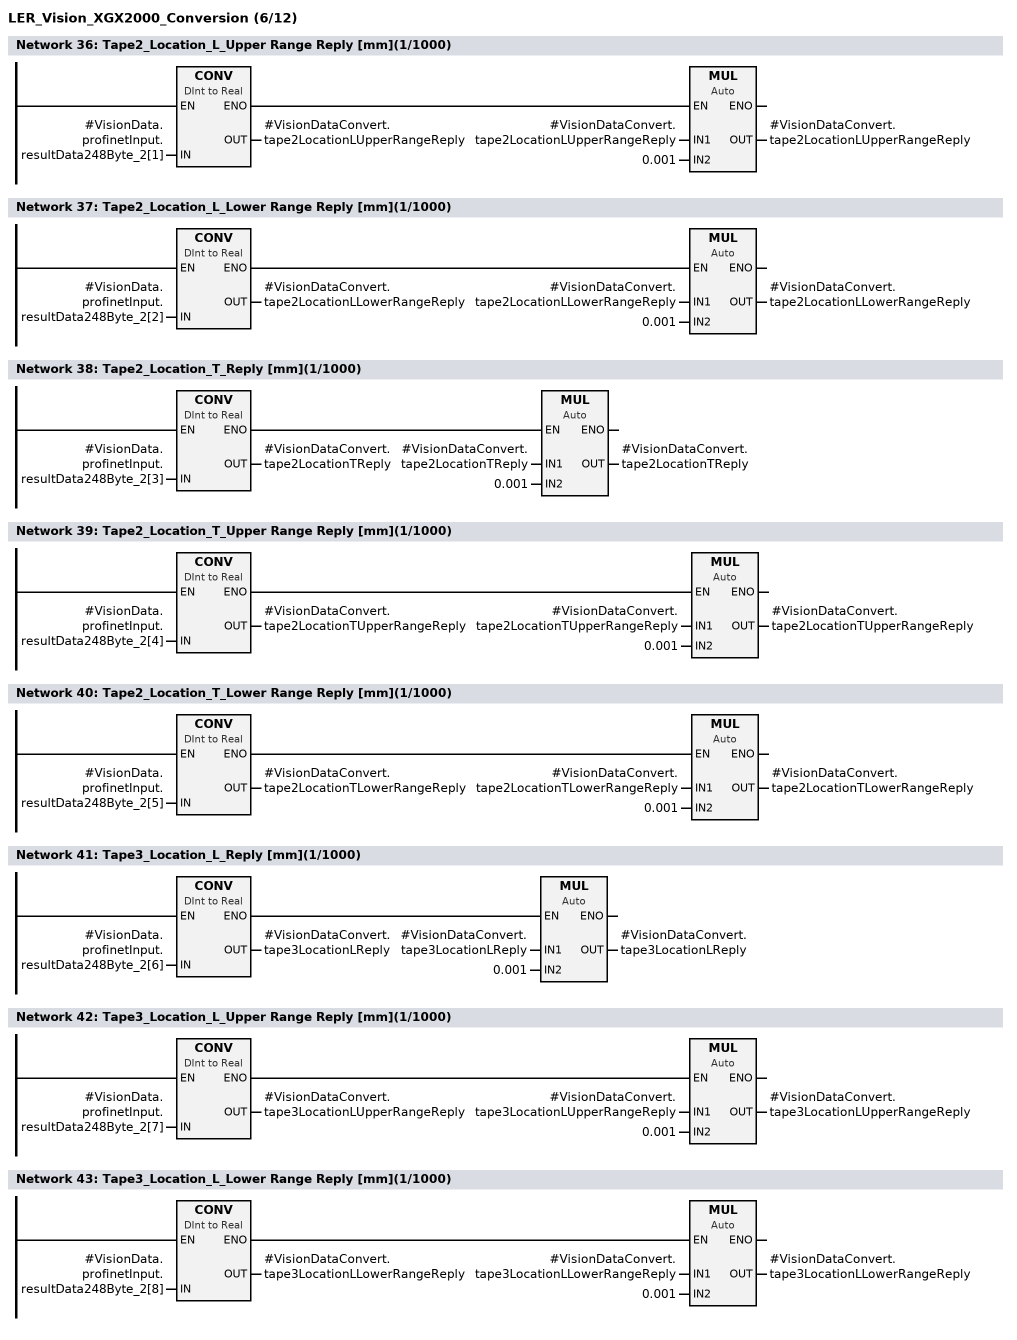
   RUNG wire#powerrail
      { S7_Templates := "[SrcType := DInt, DestType := Real]" } Convert(in := #VisionData.profinetInput.resultData248Byte_2[1], out => #VisionDataConvert.tape2LocationLUpperRangeReply)
      Mul(in1 := #VisionDataConvert.tape2LocationLUpperRangeReply, in2 := 0.001, out => #VisionDataConvert.tape2LocationLUpperRangeReply)
   END_RUNG
   // the same network as SCL:
   #VisionDataConvert.tape2LocationLUpperRangeReply := DINT_TO_REAL(#VisionData.profinetInput.resultData248Byte_2[1]);
   #VisionDataConvert.tape2LocationLUpperRangeReply := #VisionDataConvert.tape2LocationLUpperRangeReply * 0.001;
END_REGION

REGION Network 37: Tape2_Location_L_Lower Range Reply [mm](1/1000)
   RUNG wire#powerrail
      { S7_Templates := "[SrcType := DInt, DestType := Real]" } Convert(in := #VisionData.profinetInput.resultData248Byte_2[2], out => #VisionDataConvert.tape2LocationLLowerRangeReply)
      Mul(in1 := #VisionDataConvert.tape2LocationLLowerRangeReply, in2 := 0.001, out => #VisionDataConvert.tape2LocationLLowerRangeReply)
   END_RUNG
   // the same network as SCL:
   #VisionDataConvert.tape2LocationLLowerRangeReply := DINT_TO_REAL(#VisionData.profinetInput.resultData248Byte_2[2]);
   #VisionDataConvert.tape2LocationLLowerRangeReply := #VisionDataConvert.tape2LocationLLowerRangeReply * 0.001;
END_REGION

REGION Network 38: Tape2_Location_T_Reply [mm](1/1000)
   RUNG wire#powerrail
      { S7_Templates := "[SrcType := DInt, DestType := Real]" } Convert(in := #VisionData.profinetInput.resultData248Byte_2[3], out => #VisionDataConvert.tape2LocationTReply)
      Mul(in1 := #VisionDataConvert.tape2LocationTReply, in2 := 0.001, out => #VisionDataConvert.tape2LocationTReply)
   END_RUNG
   // the same network as SCL:
   #VisionDataConvert.tape2LocationTReply := DINT_TO_REAL(#VisionData.profinetInput.resultData248Byte_2[3]);
   #VisionDataConvert.tape2LocationTReply := #VisionDataConvert.tape2LocationTReply * 0.001;
END_REGION

REGION Network 39: Tape2_Location_T_Upper Range Reply [mm](1/1000)
   RUNG wire#powerrail
      { S7_Templates := "[SrcType := DInt, DestType := Real]" } Convert(in := #VisionData.profinetInput.resultData248Byte_2[4], out => #VisionDataConvert.tape2LocationTUpperRangeReply)
      Mul(in1 := #VisionDataConvert.tape2LocationTUpperRangeReply, in2 := 0.001, out => #VisionDataConvert.tape2LocationTUpperRangeReply)
   END_RUNG
   // the same network as SCL:
   #VisionDataConvert.tape2LocationTUpperRangeReply := DINT_TO_REAL(#VisionData.profinetInput.resultData248Byte_2[4]);
   #VisionDataConvert.tape2LocationTUpperRangeReply := #VisionDataConvert.tape2LocationTUpperRangeReply * 0.001;
END_REGION

REGION Network 40: Tape2_Location_T_Lower Range Reply [mm](1/1000)
   RUNG wire#powerrail
      { S7_Templates := "[SrcType := DInt, DestType := Real]" } Convert(in := #VisionData.profinetInput.resultData248Byte_2[5], out => #VisionDataConvert.tape2LocationTLowerRangeReply)
      Mul(in1 := #VisionDataConvert.tape2LocationTLowerRangeReply, in2 := 0.001, out => #VisionDataConvert.tape2LocationTLowerRangeReply)
   END_RUNG
   // the same network as SCL:
   #VisionDataConvert.tape2LocationTLowerRangeReply := DINT_TO_REAL(#VisionData.profinetInput.resultData248Byte_2[5]);
   #VisionDataConvert.tape2LocationTLowerRangeReply := #VisionDataConvert.tape2LocationTLowerRangeReply * 0.001;
END_REGION

REGION Network 41: Tape3_Location_L_Reply [mm](1/1000)
   RUNG wire#powerrail
      { S7_Templates := "[SrcType := DInt, DestType := Real]" } Convert(in := #VisionData.profinetInput.resultData248Byte_2[6], out => #VisionDataConvert.tape3LocationLReply)
      Mul(in1 := #VisionDataConvert.tape3LocationLReply, in2 := 0.001, out => #VisionDataConvert.tape3LocationLReply)
   END_RUNG
   // the same network as SCL:
   #VisionDataConvert.tape3LocationLReply := DINT_TO_REAL(#VisionData.profinetInput.resultData248Byte_2[6]);
   #VisionDataConvert.tape3LocationLReply := #VisionDataConvert.tape3LocationLReply * 0.001;
END_REGION

REGION Network 42: Tape3_Location_L_Upper Range Reply [mm](1/1000)
   RUNG wire#powerrail
      { S7_Templates := "[SrcType := DInt, DestType := Real]" } Convert(in := #VisionData.profinetInput.resultData248Byte_2[7], out => #VisionDataConvert.tape3LocationLUpperRangeReply)
      Mul(in1 := #VisionDataConvert.tape3LocationLUpperRangeReply, in2 := 0.001, out => #VisionDataConvert.tape3LocationLUpperRangeReply)
   END_RUNG
   // the same network as SCL:
   #VisionDataConvert.tape3LocationLUpperRangeReply := DINT_TO_REAL(#VisionData.profinetInput.resultData248Byte_2[7]);
   #VisionDataConvert.tape3LocationLUpperRangeReply := #VisionDataConvert.tape3LocationLUpperRangeReply * 0.001;
END_REGION

REGION Network 43: Tape3_Location_L_Lower Range Reply [mm](1/1000)
   RUNG wire#powerrail
      { S7_Templates := "[SrcType := DInt, DestType := Real]" } Convert(in := #VisionData.profinetInput.resultData248Byte_2[8], out => #VisionDataConvert.tape3LocationLLowerRangeReply)
      Mul(in1 := #VisionDataConvert.tape3LocationLLowerRangeReply, in2 := 0.001, out => #VisionDataConvert.tape3LocationLLowerRangeReply)
   END_RUNG
   // the same network as SCL:
   #VisionDataConvert.tape3LocationLLowerRangeReply := DINT_TO_REAL(#VisionData.profinetInput.resultData248Byte_2[8]);
   #VisionDataConvert.tape3LocationLLowerRangeReply := #VisionDataConvert.tape3LocationLLowerRangeReply * 0.001;
END_REGION

REGION Network 44: Tape3_Location_B_Reply [mm](1/1000)
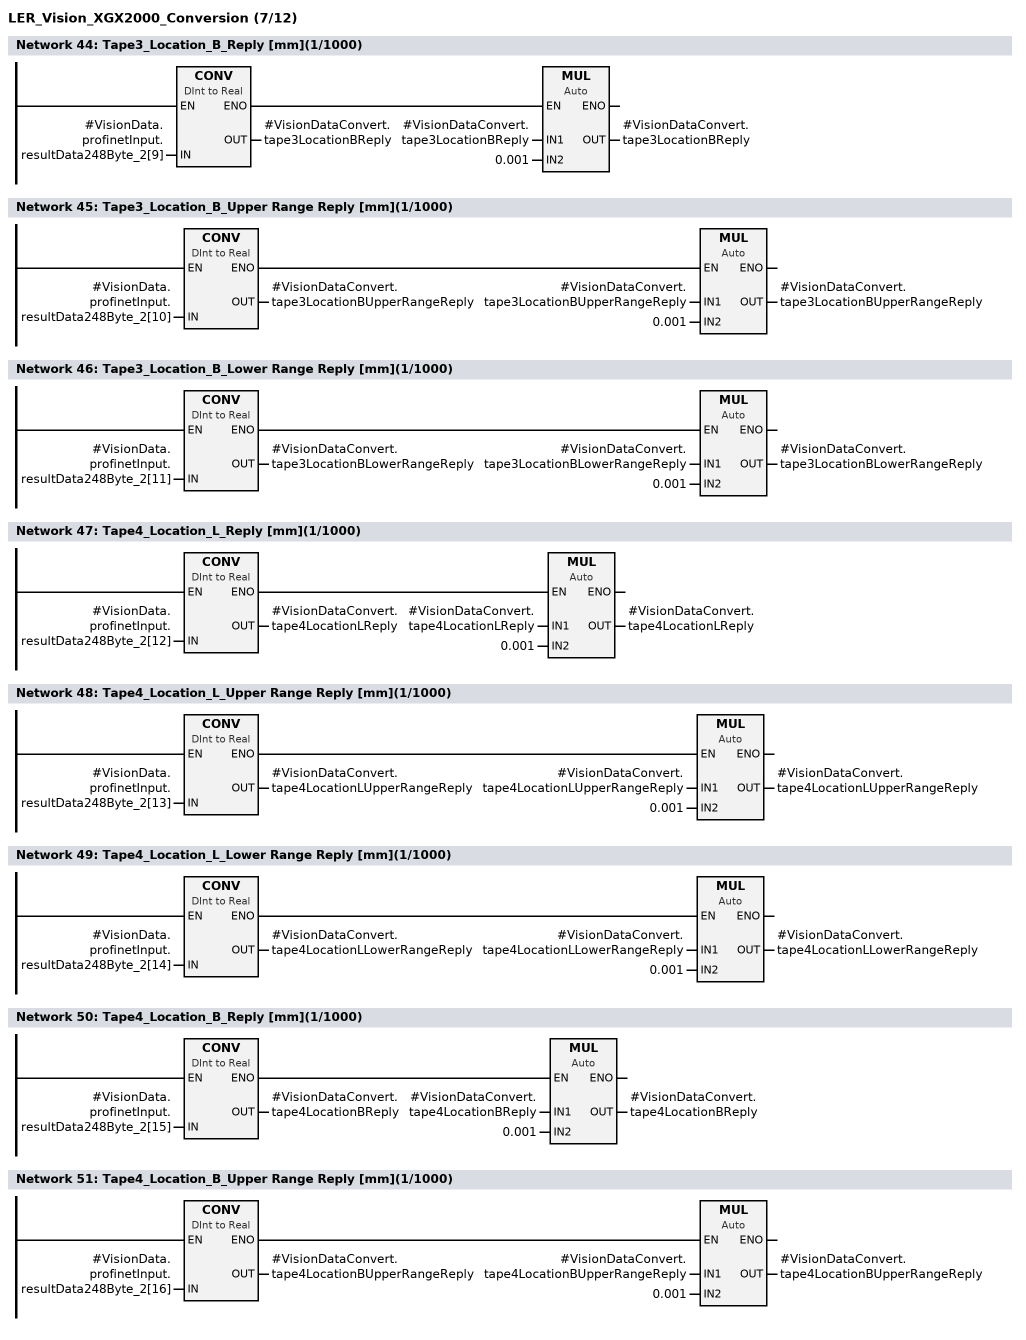
   RUNG wire#powerrail
      { S7_Templates := "[SrcType := DInt, DestType := Real]" } Convert(in := #VisionData.profinetInput.resultData248Byte_2[9], out => #VisionDataConvert.tape3LocationBReply)
      Mul(in1 := #VisionDataConvert.tape3LocationBReply, in2 := 0.001, out => #VisionDataConvert.tape3LocationBReply)
   END_RUNG
   // the same network as SCL:
   #VisionDataConvert.tape3LocationBReply := DINT_TO_REAL(#VisionData.profinetInput.resultData248Byte_2[9]);
   #VisionDataConvert.tape3LocationBReply := #VisionDataConvert.tape3LocationBReply * 0.001;
END_REGION

REGION Network 45: Tape3_Location_B_Upper Range Reply [mm](1/1000)
   RUNG wire#powerrail
      { S7_Templates := "[SrcType := DInt, DestType := Real]" } Convert(in := #VisionData.profinetInput.resultData248Byte_2[10], out => #VisionDataConvert.tape3LocationBUpperRangeReply)
      Mul(in1 := #VisionDataConvert.tape3LocationBUpperRangeReply, in2 := 0.001, out => #VisionDataConvert.tape3LocationBUpperRangeReply)
   END_RUNG
   // the same network as SCL:
   #VisionDataConvert.tape3LocationBUpperRangeReply := DINT_TO_REAL(#VisionData.profinetInput.resultData248Byte_2[10]);
   #VisionDataConvert.tape3LocationBUpperRangeReply := #VisionDataConvert.tape3LocationBUpperRangeReply * 0.001;
END_REGION

REGION Network 46: Tape3_Location_B_Lower Range Reply [mm](1/1000)
   RUNG wire#powerrail
      { S7_Templates := "[SrcType := DInt, DestType := Real]" } Convert(in := #VisionData.profinetInput.resultData248Byte_2[11], out => #VisionDataConvert.tape3LocationBLowerRangeReply)
      Mul(in1 := #VisionDataConvert.tape3LocationBLowerRangeReply, in2 := 0.001, out => #VisionDataConvert.tape3LocationBLowerRangeReply)
   END_RUNG
   // the same network as SCL:
   #VisionDataConvert.tape3LocationBLowerRangeReply := DINT_TO_REAL(#VisionData.profinetInput.resultData248Byte_2[11]);
   #VisionDataConvert.tape3LocationBLowerRangeReply := #VisionDataConvert.tape3LocationBLowerRangeReply * 0.001;
END_REGION

REGION Network 47: Tape4_Location_L_Reply [mm](1/1000)
   RUNG wire#powerrail
      { S7_Templates := "[SrcType := DInt, DestType := Real]" } Convert(in := #VisionData.profinetInput.resultData248Byte_2[12], out => #VisionDataConvert.tape4LocationLReply)
      Mul(in1 := #VisionDataConvert.tape4LocationLReply, in2 := 0.001, out => #VisionDataConvert.tape4LocationLReply)
   END_RUNG
   // the same network as SCL:
   #VisionDataConvert.tape4LocationLReply := DINT_TO_REAL(#VisionData.profinetInput.resultData248Byte_2[12]);
   #VisionDataConvert.tape4LocationLReply := #VisionDataConvert.tape4LocationLReply * 0.001;
END_REGION

REGION Network 48: Tape4_Location_L_Upper Range Reply [mm](1/1000)
   RUNG wire#powerrail
      { S7_Templates := "[SrcType := DInt, DestType := Real]" } Convert(in := #VisionData.profinetInput.resultData248Byte_2[13], out => #VisionDataConvert.tape4LocationLUpperRangeReply)
      Mul(in1 := #VisionDataConvert.tape4LocationLUpperRangeReply, in2 := 0.001, out => #VisionDataConvert.tape4LocationLUpperRangeReply)
   END_RUNG
   // the same network as SCL:
   #VisionDataConvert.tape4LocationLUpperRangeReply := DINT_TO_REAL(#VisionData.profinetInput.resultData248Byte_2[13]);
   #VisionDataConvert.tape4LocationLUpperRangeReply := #VisionDataConvert.tape4LocationLUpperRangeReply * 0.001;
END_REGION

REGION Network 49: Tape4_Location_L_Lower Range Reply [mm](1/1000)
   RUNG wire#powerrail
      { S7_Templates := "[SrcType := DInt, DestType := Real]" } Convert(in := #VisionData.profinetInput.resultData248Byte_2[14], out => #VisionDataConvert.tape4LocationLLowerRangeReply)
      Mul(in1 := #VisionDataConvert.tape4LocationLLowerRangeReply, in2 := 0.001, out => #VisionDataConvert.tape4LocationLLowerRangeReply)
   END_RUNG
   // the same network as SCL:
   #VisionDataConvert.tape4LocationLLowerRangeReply := DINT_TO_REAL(#VisionData.profinetInput.resultData248Byte_2[14]);
   #VisionDataConvert.tape4LocationLLowerRangeReply := #VisionDataConvert.tape4LocationLLowerRangeReply * 0.001;
END_REGION

REGION Network 50: Tape4_Location_B_Reply [mm](1/1000)
   RUNG wire#powerrail
      { S7_Templates := "[SrcType := DInt, DestType := Real]" } Convert(in := #VisionData.profinetInput.resultData248Byte_2[15], out => #VisionDataConvert.tape4LocationBReply)
      Mul(in1 := #VisionDataConvert.tape4LocationBReply, in2 := 0.001, out => #VisionDataConvert.tape4LocationBReply)
   END_RUNG
   // the same network as SCL:
   #VisionDataConvert.tape4LocationBReply := DINT_TO_REAL(#VisionData.profinetInput.resultData248Byte_2[15]);
   #VisionDataConvert.tape4LocationBReply := #VisionDataConvert.tape4LocationBReply * 0.001;
END_REGION

REGION Network 51: Tape4_Location_B_Upper Range Reply [mm](1/1000)
   RUNG wire#powerrail
      { S7_Templates := "[SrcType := DInt, DestType := Real]" } Convert(in := #VisionData.profinetInput.resultData248Byte_2[16], out => #VisionDataConvert.tape4LocationBUpperRangeReply)
      Mul(in1 := #VisionDataConvert.tape4LocationBUpperRangeReply, in2 := 0.001, out => #VisionDataConvert.tape4LocationBUpperRangeReply)
   END_RUNG
   // the same network as SCL:
   #VisionDataConvert.tape4LocationBUpperRangeReply := DINT_TO_REAL(#VisionData.profinetInput.resultData248Byte_2[16]);
   #VisionDataConvert.tape4LocationBUpperRangeReply := #VisionDataConvert.tape4LocationBUpperRangeReply * 0.001;
END_REGION

REGION Network 52: Tape4_Location_B_Lower Range Reply [mm](1/1000)
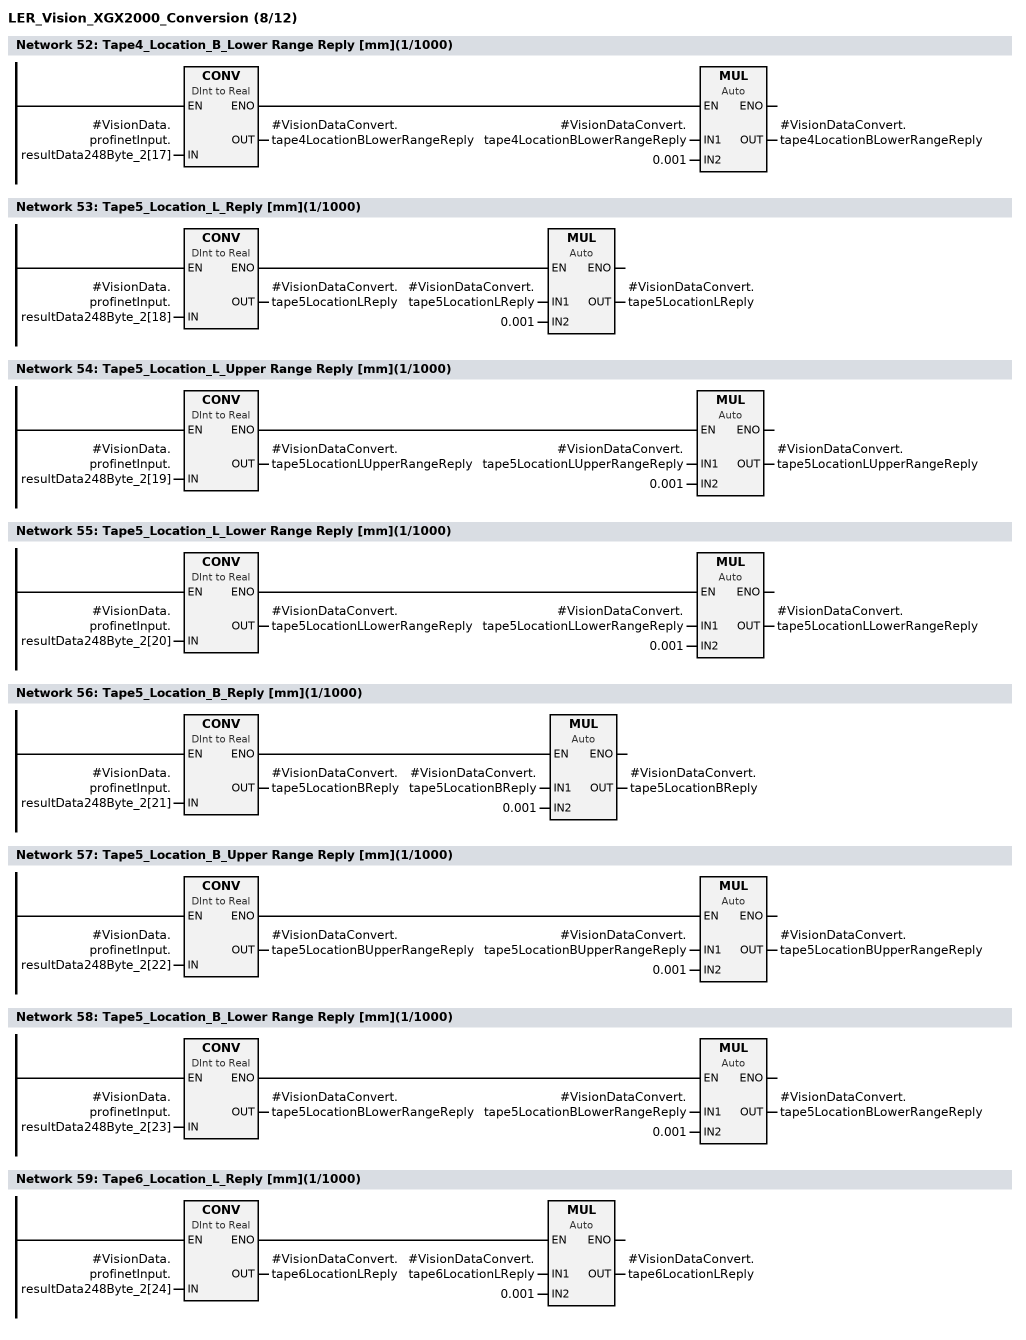
   RUNG wire#powerrail
      { S7_Templates := "[SrcType := DInt, DestType := Real]" } Convert(in := #VisionData.profinetInput.resultData248Byte_2[17], out => #VisionDataConvert.tape4LocationBLowerRangeReply)
      Mul(in1 := #VisionDataConvert.tape4LocationBLowerRangeReply, in2 := 0.001, out => #VisionDataConvert.tape4LocationBLowerRangeReply)
   END_RUNG
   // the same network as SCL:
   #VisionDataConvert.tape4LocationBLowerRangeReply := DINT_TO_REAL(#VisionData.profinetInput.resultData248Byte_2[17]);
   #VisionDataConvert.tape4LocationBLowerRangeReply := #VisionDataConvert.tape4LocationBLowerRangeReply * 0.001;
END_REGION

REGION Network 53: Tape5_Location_L_Reply [mm](1/1000)
   RUNG wire#powerrail
      { S7_Templates := "[SrcType := DInt, DestType := Real]" } Convert(in := #VisionData.profinetInput.resultData248Byte_2[18], out => #VisionDataConvert.tape5LocationLReply)
      Mul(in1 := #VisionDataConvert.tape5LocationLReply, in2 := 0.001, out => #VisionDataConvert.tape5LocationLReply)
   END_RUNG
   // the same network as SCL:
   #VisionDataConvert.tape5LocationLReply := DINT_TO_REAL(#VisionData.profinetInput.resultData248Byte_2[18]);
   #VisionDataConvert.tape5LocationLReply := #VisionDataConvert.tape5LocationLReply * 0.001;
END_REGION

REGION Network 54: Tape5_Location_L_Upper Range Reply [mm](1/1000)
   RUNG wire#powerrail
      { S7_Templates := "[SrcType := DInt, DestType := Real]" } Convert(in := #VisionData.profinetInput.resultData248Byte_2[19], out => #VisionDataConvert.tape5LocationLUpperRangeReply)
      Mul(in1 := #VisionDataConvert.tape5LocationLUpperRangeReply, in2 := 0.001, out => #VisionDataConvert.tape5LocationLUpperRangeReply)
   END_RUNG
   // the same network as SCL:
   #VisionDataConvert.tape5LocationLUpperRangeReply := DINT_TO_REAL(#VisionData.profinetInput.resultData248Byte_2[19]);
   #VisionDataConvert.tape5LocationLUpperRangeReply := #VisionDataConvert.tape5LocationLUpperRangeReply * 0.001;
END_REGION

REGION Network 55: Tape5_Location_L_Lower Range Reply [mm](1/1000)
   RUNG wire#powerrail
      { S7_Templates := "[SrcType := DInt, DestType := Real]" } Convert(in := #VisionData.profinetInput.resultData248Byte_2[20], out => #VisionDataConvert.tape5LocationLLowerRangeReply)
      Mul(in1 := #VisionDataConvert.tape5LocationLLowerRangeReply, in2 := 0.001, out => #VisionDataConvert.tape5LocationLLowerRangeReply)
   END_RUNG
   // the same network as SCL:
   #VisionDataConvert.tape5LocationLLowerRangeReply := DINT_TO_REAL(#VisionData.profinetInput.resultData248Byte_2[20]);
   #VisionDataConvert.tape5LocationLLowerRangeReply := #VisionDataConvert.tape5LocationLLowerRangeReply * 0.001;
END_REGION

REGION Network 56: Tape5_Location_B_Reply [mm](1/1000)
   RUNG wire#powerrail
      { S7_Templates := "[SrcType := DInt, DestType := Real]" } Convert(in := #VisionData.profinetInput.resultData248Byte_2[21], out => #VisionDataConvert.tape5LocationBReply)
      Mul(in1 := #VisionDataConvert.tape5LocationBReply, in2 := 0.001, out => #VisionDataConvert.tape5LocationBReply)
   END_RUNG
   // the same network as SCL:
   #VisionDataConvert.tape5LocationBReply := DINT_TO_REAL(#VisionData.profinetInput.resultData248Byte_2[21]);
   #VisionDataConvert.tape5LocationBReply := #VisionDataConvert.tape5LocationBReply * 0.001;
END_REGION

REGION Network 57: Tape5_Location_B_Upper Range Reply [mm](1/1000)
   RUNG wire#powerrail
      { S7_Templates := "[SrcType := DInt, DestType := Real]" } Convert(in := #VisionData.profinetInput.resultData248Byte_2[22], out => #VisionDataConvert.tape5LocationBUpperRangeReply)
      Mul(in1 := #VisionDataConvert.tape5LocationBUpperRangeReply, in2 := 0.001, out => #VisionDataConvert.tape5LocationBUpperRangeReply)
   END_RUNG
   // the same network as SCL:
   #VisionDataConvert.tape5LocationBUpperRangeReply := DINT_TO_REAL(#VisionData.profinetInput.resultData248Byte_2[22]);
   #VisionDataConvert.tape5LocationBUpperRangeReply := #VisionDataConvert.tape5LocationBUpperRangeReply * 0.001;
END_REGION

REGION Network 58: Tape5_Location_B_Lower Range Reply [mm](1/1000)
   RUNG wire#powerrail
      { S7_Templates := "[SrcType := DInt, DestType := Real]" } Convert(in := #VisionData.profinetInput.resultData248Byte_2[23], out => #VisionDataConvert.tape5LocationBLowerRangeReply)
      Mul(in1 := #VisionDataConvert.tape5LocationBLowerRangeReply, in2 := 0.001, out => #VisionDataConvert.tape5LocationBLowerRangeReply)
   END_RUNG
   // the same network as SCL:
   #VisionDataConvert.tape5LocationBLowerRangeReply := DINT_TO_REAL(#VisionData.profinetInput.resultData248Byte_2[23]);
   #VisionDataConvert.tape5LocationBLowerRangeReply := #VisionDataConvert.tape5LocationBLowerRangeReply * 0.001;
END_REGION

REGION Network 59: Tape6_Location_L_Reply [mm](1/1000)
   RUNG wire#powerrail
      { S7_Templates := "[SrcType := DInt, DestType := Real]" } Convert(in := #VisionData.profinetInput.resultData248Byte_2[24], out => #VisionDataConvert.tape6LocationLReply)
      Mul(in1 := #VisionDataConvert.tape6LocationLReply, in2 := 0.001, out => #VisionDataConvert.tape6LocationLReply)
   END_RUNG
   // the same network as SCL:
   #VisionDataConvert.tape6LocationLReply := DINT_TO_REAL(#VisionData.profinetInput.resultData248Byte_2[24]);
   #VisionDataConvert.tape6LocationLReply := #VisionDataConvert.tape6LocationLReply * 0.001;
END_REGION

REGION Network 60: Tape6_Location_L_Upper Range Reply [mm](1/1000)
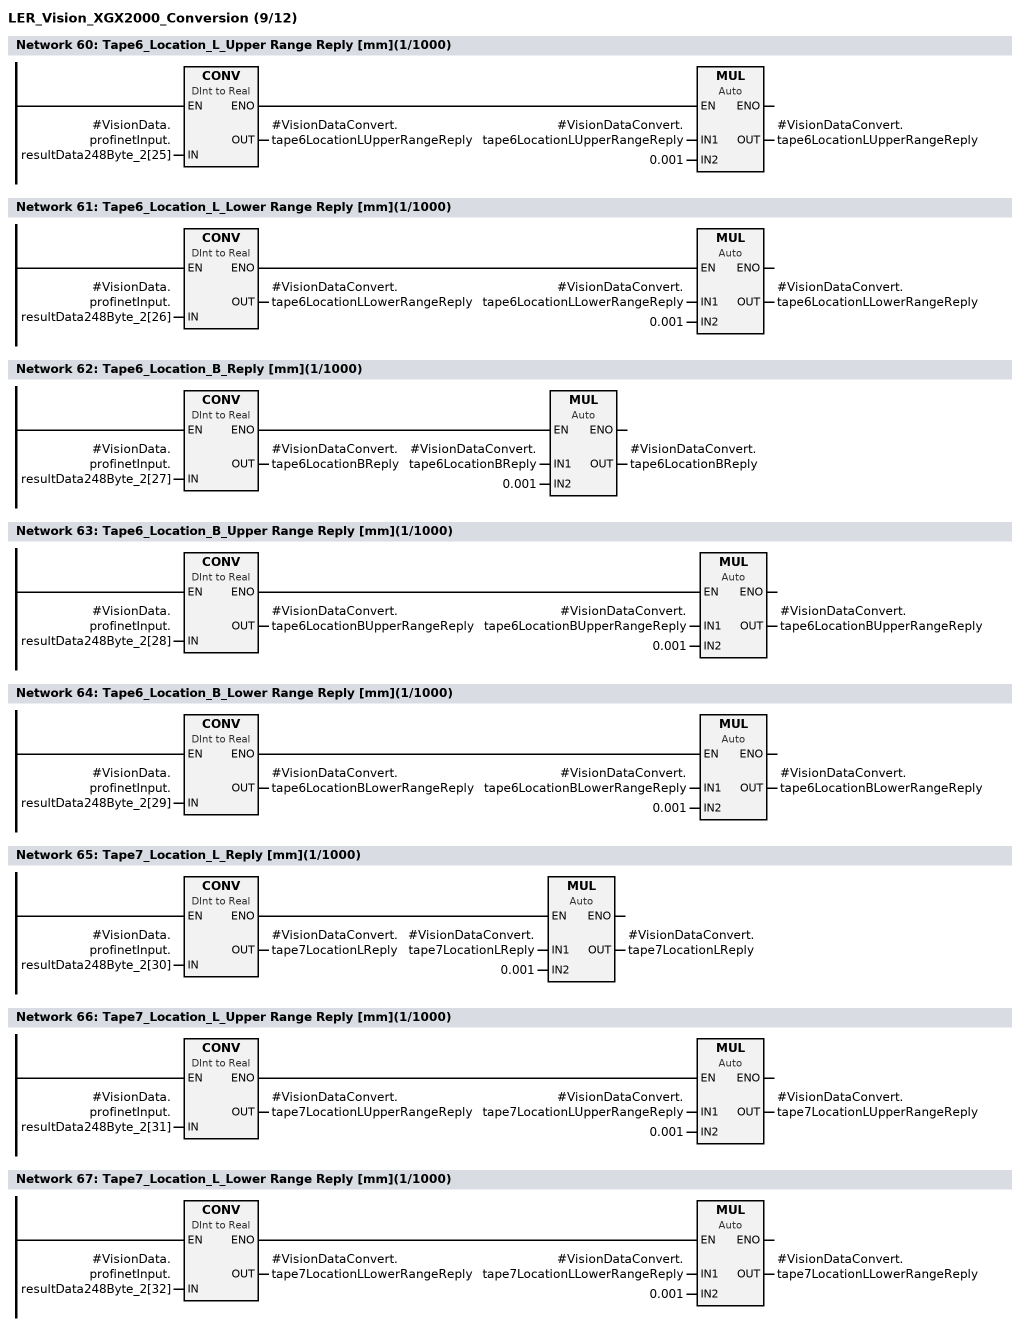
   RUNG wire#powerrail
      { S7_Templates := "[SrcType := DInt, DestType := Real]" } Convert(in := #VisionData.profinetInput.resultData248Byte_2[25], out => #VisionDataConvert.tape6LocationLUpperRangeReply)
      Mul(in1 := #VisionDataConvert.tape6LocationLUpperRangeReply, in2 := 0.001, out => #VisionDataConvert.tape6LocationLUpperRangeReply)
   END_RUNG
   // the same network as SCL:
   #VisionDataConvert.tape6LocationLUpperRangeReply := DINT_TO_REAL(#VisionData.profinetInput.resultData248Byte_2[25]);
   #VisionDataConvert.tape6LocationLUpperRangeReply := #VisionDataConvert.tape6LocationLUpperRangeReply * 0.001;
END_REGION

REGION Network 61: Tape6_Location_L_Lower Range Reply [mm](1/1000)
   RUNG wire#powerrail
      { S7_Templates := "[SrcType := DInt, DestType := Real]" } Convert(in := #VisionData.profinetInput.resultData248Byte_2[26], out => #VisionDataConvert.tape6LocationLLowerRangeReply)
      Mul(in1 := #VisionDataConvert.tape6LocationLLowerRangeReply, in2 := 0.001, out => #VisionDataConvert.tape6LocationLLowerRangeReply)
   END_RUNG
   // the same network as SCL:
   #VisionDataConvert.tape6LocationLLowerRangeReply := DINT_TO_REAL(#VisionData.profinetInput.resultData248Byte_2[26]);
   #VisionDataConvert.tape6LocationLLowerRangeReply := #VisionDataConvert.tape6LocationLLowerRangeReply * 0.001;
END_REGION

REGION Network 62: Tape6_Location_B_Reply [mm](1/1000)
   RUNG wire#powerrail
      { S7_Templates := "[SrcType := DInt, DestType := Real]" } Convert(in := #VisionData.profinetInput.resultData248Byte_2[27], out => #VisionDataConvert.tape6LocationBReply)
      Mul(in1 := #VisionDataConvert.tape6LocationBReply, in2 := 0.001, out => #VisionDataConvert.tape6LocationBReply)
   END_RUNG
   // the same network as SCL:
   #VisionDataConvert.tape6LocationBReply := DINT_TO_REAL(#VisionData.profinetInput.resultData248Byte_2[27]);
   #VisionDataConvert.tape6LocationBReply := #VisionDataConvert.tape6LocationBReply * 0.001;
END_REGION

REGION Network 63: Tape6_Location_B_Upper Range Reply [mm](1/1000)
   RUNG wire#powerrail
      { S7_Templates := "[SrcType := DInt, DestType := Real]" } Convert(in := #VisionData.profinetInput.resultData248Byte_2[28], out => #VisionDataConvert.tape6LocationBUpperRangeReply)
      Mul(in1 := #VisionDataConvert.tape6LocationBUpperRangeReply, in2 := 0.001, out => #VisionDataConvert.tape6LocationBUpperRangeReply)
   END_RUNG
   // the same network as SCL:
   #VisionDataConvert.tape6LocationBUpperRangeReply := DINT_TO_REAL(#VisionData.profinetInput.resultData248Byte_2[28]);
   #VisionDataConvert.tape6LocationBUpperRangeReply := #VisionDataConvert.tape6LocationBUpperRangeReply * 0.001;
END_REGION

REGION Network 64: Tape6_Location_B_Lower Range Reply [mm](1/1000)
   RUNG wire#powerrail
      { S7_Templates := "[SrcType := DInt, DestType := Real]" } Convert(in := #VisionData.profinetInput.resultData248Byte_2[29], out => #VisionDataConvert.tape6LocationBLowerRangeReply)
      Mul(in1 := #VisionDataConvert.tape6LocationBLowerRangeReply, in2 := 0.001, out => #VisionDataConvert.tape6LocationBLowerRangeReply)
   END_RUNG
   // the same network as SCL:
   #VisionDataConvert.tape6LocationBLowerRangeReply := DINT_TO_REAL(#VisionData.profinetInput.resultData248Byte_2[29]);
   #VisionDataConvert.tape6LocationBLowerRangeReply := #VisionDataConvert.tape6LocationBLowerRangeReply * 0.001;
END_REGION

REGION Network 65: Tape7_Location_L_Reply [mm](1/1000)
   RUNG wire#powerrail
      { S7_Templates := "[SrcType := DInt, DestType := Real]" } Convert(in := #VisionData.profinetInput.resultData248Byte_2[30], out => #VisionDataConvert.tape7LocationLReply)
      Mul(in1 := #VisionDataConvert.tape7LocationLReply, in2 := 0.001, out => #VisionDataConvert.tape7LocationLReply)
   END_RUNG
   // the same network as SCL:
   #VisionDataConvert.tape7LocationLReply := DINT_TO_REAL(#VisionData.profinetInput.resultData248Byte_2[30]);
   #VisionDataConvert.tape7LocationLReply := #VisionDataConvert.tape7LocationLReply * 0.001;
END_REGION

REGION Network 66: Tape7_Location_L_Upper Range Reply [mm](1/1000)
   RUNG wire#powerrail
      { S7_Templates := "[SrcType := DInt, DestType := Real]" } Convert(in := #VisionData.profinetInput.resultData248Byte_2[31], out => #VisionDataConvert.tape7LocationLUpperRangeReply)
      Mul(in1 := #VisionDataConvert.tape7LocationLUpperRangeReply, in2 := 0.001, out => #VisionDataConvert.tape7LocationLUpperRangeReply)
   END_RUNG
   // the same network as SCL:
   #VisionDataConvert.tape7LocationLUpperRangeReply := DINT_TO_REAL(#VisionData.profinetInput.resultData248Byte_2[31]);
   #VisionDataConvert.tape7LocationLUpperRangeReply := #VisionDataConvert.tape7LocationLUpperRangeReply * 0.001;
END_REGION

REGION Network 67: Tape7_Location_L_Lower Range Reply [mm](1/1000)
   RUNG wire#powerrail
      { S7_Templates := "[SrcType := DInt, DestType := Real]" } Convert(in := #VisionData.profinetInput.resultData248Byte_2[32], out => #VisionDataConvert.tape7LocationLLowerRangeReply)
      Mul(in1 := #VisionDataConvert.tape7LocationLLowerRangeReply, in2 := 0.001, out => #VisionDataConvert.tape7LocationLLowerRangeReply)
   END_RUNG
   // the same network as SCL:
   #VisionDataConvert.tape7LocationLLowerRangeReply := DINT_TO_REAL(#VisionData.profinetInput.resultData248Byte_2[32]);
   #VisionDataConvert.tape7LocationLLowerRangeReply := #VisionDataConvert.tape7LocationLLowerRangeReply * 0.001;
END_REGION

REGION Network 68: Tape7_Location_T_Reply [mm](1/1000)
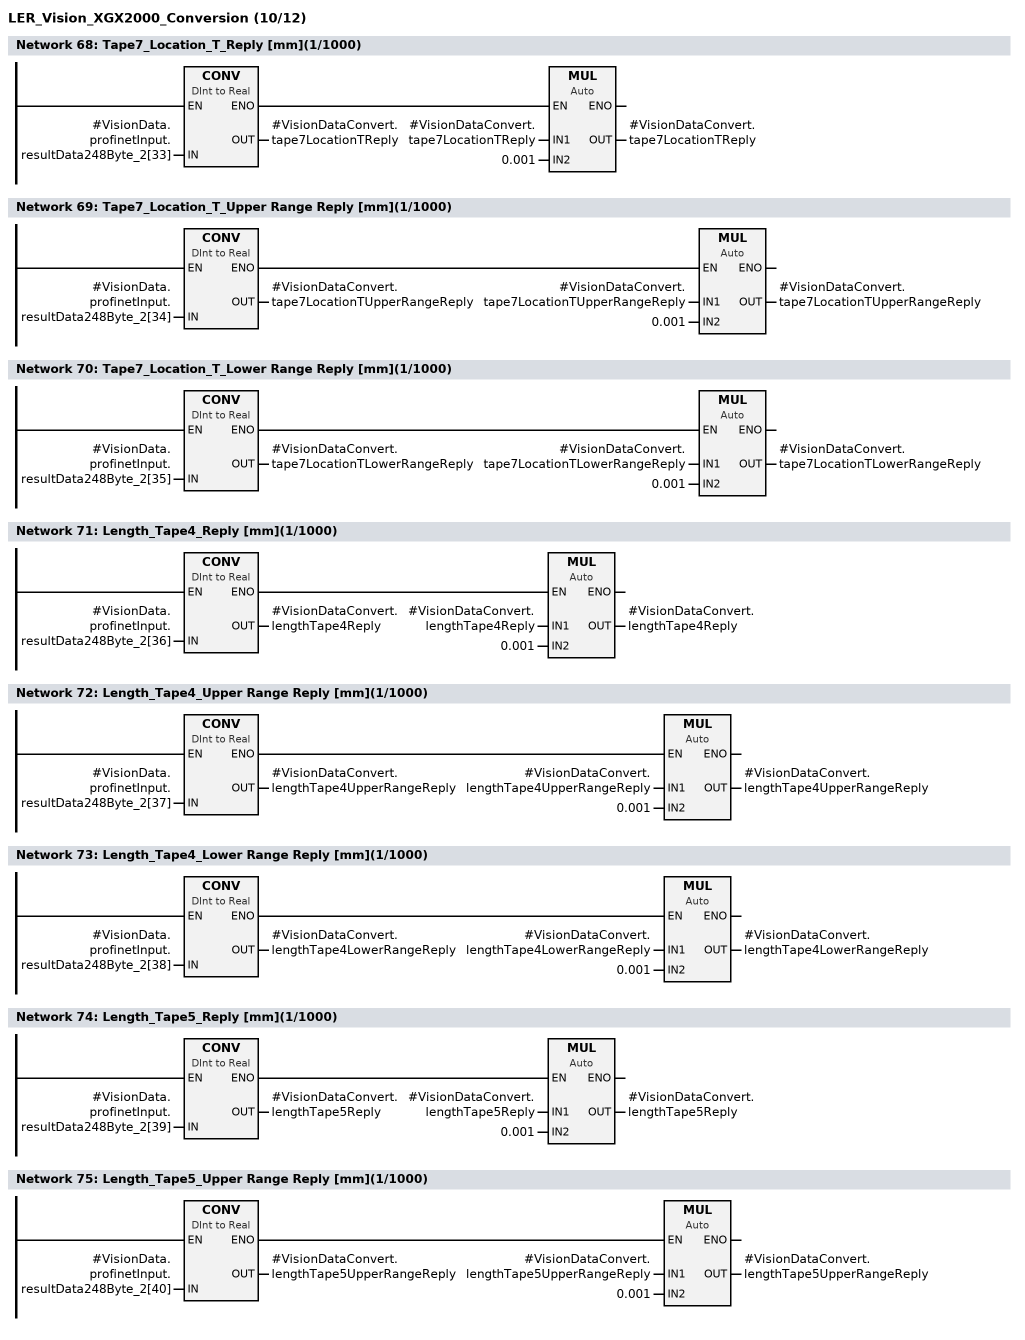
   RUNG wire#powerrail
      { S7_Templates := "[SrcType := DInt, DestType := Real]" } Convert(in := #VisionData.profinetInput.resultData248Byte_2[33], out => #VisionDataConvert.tape7LocationTReply)
      Mul(in1 := #VisionDataConvert.tape7LocationTReply, in2 := 0.001, out => #VisionDataConvert.tape7LocationTReply)
   END_RUNG
   // the same network as SCL:
   #VisionDataConvert.tape7LocationTReply := DINT_TO_REAL(#VisionData.profinetInput.resultData248Byte_2[33]);
   #VisionDataConvert.tape7LocationTReply := #VisionDataConvert.tape7LocationTReply * 0.001;
END_REGION

REGION Network 69: Tape7_Location_T_Upper Range Reply [mm](1/1000)
   RUNG wire#powerrail
      { S7_Templates := "[SrcType := DInt, DestType := Real]" } Convert(in := #VisionData.profinetInput.resultData248Byte_2[34], out => #VisionDataConvert.tape7LocationTUpperRangeReply)
      Mul(in1 := #VisionDataConvert.tape7LocationTUpperRangeReply, in2 := 0.001, out => #VisionDataConvert.tape7LocationTUpperRangeReply)
   END_RUNG
   // the same network as SCL:
   #VisionDataConvert.tape7LocationTUpperRangeReply := DINT_TO_REAL(#VisionData.profinetInput.resultData248Byte_2[34]);
   #VisionDataConvert.tape7LocationTUpperRangeReply := #VisionDataConvert.tape7LocationTUpperRangeReply * 0.001;
END_REGION

REGION Network 70: Tape7_Location_T_Lower Range Reply [mm](1/1000)
   RUNG wire#powerrail
      { S7_Templates := "[SrcType := DInt, DestType := Real]" } Convert(in := #VisionData.profinetInput.resultData248Byte_2[35], out => #VisionDataConvert.tape7LocationTLowerRangeReply)
      Mul(in1 := #VisionDataConvert.tape7LocationTLowerRangeReply, in2 := 0.001, out => #VisionDataConvert.tape7LocationTLowerRangeReply)
   END_RUNG
   // the same network as SCL:
   #VisionDataConvert.tape7LocationTLowerRangeReply := DINT_TO_REAL(#VisionData.profinetInput.resultData248Byte_2[35]);
   #VisionDataConvert.tape7LocationTLowerRangeReply := #VisionDataConvert.tape7LocationTLowerRangeReply * 0.001;
END_REGION

REGION Network 71: Length_Tape4_Reply [mm](1/1000)
   RUNG wire#powerrail
      { S7_Templates := "[SrcType := DInt, DestType := Real]" } Convert(in := #VisionData.profinetInput.resultData248Byte_2[36], out => #VisionDataConvert.lengthTape4Reply)
      Mul(in1 := #VisionDataConvert.lengthTape4Reply, in2 := 0.001, out => #VisionDataConvert.lengthTape4Reply)
   END_RUNG
   // the same network as SCL:
   #VisionDataConvert.lengthTape4Reply := DINT_TO_REAL(#VisionData.profinetInput.resultData248Byte_2[36]);
   #VisionDataConvert.lengthTape4Reply := #VisionDataConvert.lengthTape4Reply * 0.001;
END_REGION

REGION Network 72: Length_Tape4_Upper Range Reply [mm](1/1000)
   RUNG wire#powerrail
      { S7_Templates := "[SrcType := DInt, DestType := Real]" } Convert(in := #VisionData.profinetInput.resultData248Byte_2[37], out => #VisionDataConvert.lengthTape4UpperRangeReply)
      Mul(in1 := #VisionDataConvert.lengthTape4UpperRangeReply, in2 := 0.001, out => #VisionDataConvert.lengthTape4UpperRangeReply)
   END_RUNG
   // the same network as SCL:
   #VisionDataConvert.lengthTape4UpperRangeReply := DINT_TO_REAL(#VisionData.profinetInput.resultData248Byte_2[37]);
   #VisionDataConvert.lengthTape4UpperRangeReply := #VisionDataConvert.lengthTape4UpperRangeReply * 0.001;
END_REGION

REGION Network 73: Length_Tape4_Lower Range Reply [mm](1/1000)
   RUNG wire#powerrail
      { S7_Templates := "[SrcType := DInt, DestType := Real]" } Convert(in := #VisionData.profinetInput.resultData248Byte_2[38], out => #VisionDataConvert.lengthTape4LowerRangeReply)
      Mul(in1 := #VisionDataConvert.lengthTape4LowerRangeReply, in2 := 0.001, out => #VisionDataConvert.lengthTape4LowerRangeReply)
   END_RUNG
   // the same network as SCL:
   #VisionDataConvert.lengthTape4LowerRangeReply := DINT_TO_REAL(#VisionData.profinetInput.resultData248Byte_2[38]);
   #VisionDataConvert.lengthTape4LowerRangeReply := #VisionDataConvert.lengthTape4LowerRangeReply * 0.001;
END_REGION

REGION Network 74: Length_Tape5_Reply [mm](1/1000)
   RUNG wire#powerrail
      { S7_Templates := "[SrcType := DInt, DestType := Real]" } Convert(in := #VisionData.profinetInput.resultData248Byte_2[39], out => #VisionDataConvert.lengthTape5Reply)
      Mul(in1 := #VisionDataConvert.lengthTape5Reply, in2 := 0.001, out => #VisionDataConvert.lengthTape5Reply)
   END_RUNG
   // the same network as SCL:
   #VisionDataConvert.lengthTape5Reply := DINT_TO_REAL(#VisionData.profinetInput.resultData248Byte_2[39]);
   #VisionDataConvert.lengthTape5Reply := #VisionDataConvert.lengthTape5Reply * 0.001;
END_REGION

REGION Network 75: Length_Tape5_Upper Range Reply [mm](1/1000)
   RUNG wire#powerrail
      { S7_Templates := "[SrcType := DInt, DestType := Real]" } Convert(in := #VisionData.profinetInput.resultData248Byte_2[40], out => #VisionDataConvert.lengthTape5UpperRangeReply)
      Mul(in1 := #VisionDataConvert.lengthTape5UpperRangeReply, in2 := 0.001, out => #VisionDataConvert.lengthTape5UpperRangeReply)
   END_RUNG
   // the same network as SCL:
   #VisionDataConvert.lengthTape5UpperRangeReply := DINT_TO_REAL(#VisionData.profinetInput.resultData248Byte_2[40]);
   #VisionDataConvert.lengthTape5UpperRangeReply := #VisionDataConvert.lengthTape5UpperRangeReply * 0.001;
END_REGION

REGION Network 76: Length_Tape5_Lower Range Reply [mm](1/1000)
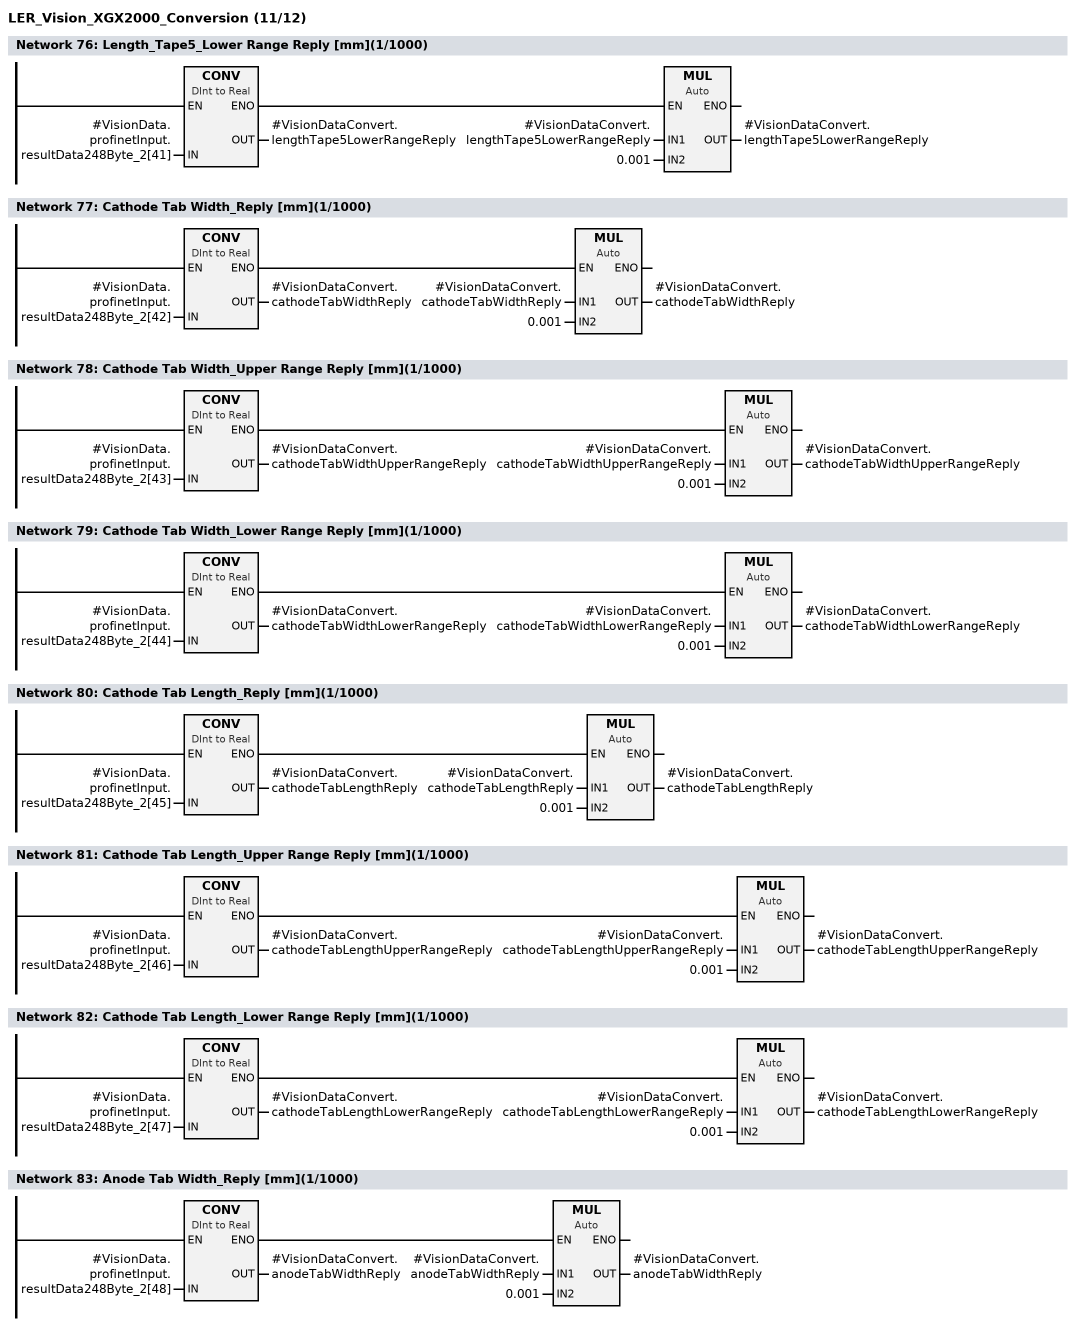
   RUNG wire#powerrail
      { S7_Templates := "[SrcType := DInt, DestType := Real]" } Convert(in := #VisionData.profinetInput.resultData248Byte_2[41], out => #VisionDataConvert.lengthTape5LowerRangeReply)
      Mul(in1 := #VisionDataConvert.lengthTape5LowerRangeReply, in2 := 0.001, out => #VisionDataConvert.lengthTape5LowerRangeReply)
   END_RUNG
   // the same network as SCL:
   #VisionDataConvert.lengthTape5LowerRangeReply := DINT_TO_REAL(#VisionData.profinetInput.resultData248Byte_2[41]);
   #VisionDataConvert.lengthTape5LowerRangeReply := #VisionDataConvert.lengthTape5LowerRangeReply * 0.001;
END_REGION

REGION Network 77: Cathode Tab Width_Reply [mm](1/1000)
   RUNG wire#powerrail
      { S7_Templates := "[SrcType := DInt, DestType := Real]" } Convert(in := #VisionData.profinetInput.resultData248Byte_2[42], out => #VisionDataConvert.cathodeTabWidthReply)
      Mul(in1 := #VisionDataConvert.cathodeTabWidthReply, in2 := 0.001, out => #VisionDataConvert.cathodeTabWidthReply)
   END_RUNG
   // the same network as SCL:
   #VisionDataConvert.cathodeTabWidthReply := DINT_TO_REAL(#VisionData.profinetInput.resultData248Byte_2[42]);
   #VisionDataConvert.cathodeTabWidthReply := #VisionDataConvert.cathodeTabWidthReply * 0.001;
END_REGION

REGION Network 78: Cathode Tab Width_Upper Range Reply [mm](1/1000)
   RUNG wire#powerrail
      { S7_Templates := "[SrcType := DInt, DestType := Real]" } Convert(in := #VisionData.profinetInput.resultData248Byte_2[43], out => #VisionDataConvert.cathodeTabWidthUpperRangeReply)
      Mul(in1 := #VisionDataConvert.cathodeTabWidthUpperRangeReply, in2 := 0.001, out => #VisionDataConvert.cathodeTabWidthUpperRangeReply)
   END_RUNG
   // the same network as SCL:
   #VisionDataConvert.cathodeTabWidthUpperRangeReply := DINT_TO_REAL(#VisionData.profinetInput.resultData248Byte_2[43]);
   #VisionDataConvert.cathodeTabWidthUpperRangeReply := #VisionDataConvert.cathodeTabWidthUpperRangeReply * 0.001;
END_REGION

REGION Network 79: Cathode Tab Width_Lower Range Reply [mm](1/1000)
   RUNG wire#powerrail
      { S7_Templates := "[SrcType := DInt, DestType := Real]" } Convert(in := #VisionData.profinetInput.resultData248Byte_2[44], out => #VisionDataConvert.cathodeTabWidthLowerRangeReply)
      Mul(in1 := #VisionDataConvert.cathodeTabWidthLowerRangeReply, in2 := 0.001, out => #VisionDataConvert.cathodeTabWidthLowerRangeReply)
   END_RUNG
   // the same network as SCL:
   #VisionDataConvert.cathodeTabWidthLowerRangeReply := DINT_TO_REAL(#VisionData.profinetInput.resultData248Byte_2[44]);
   #VisionDataConvert.cathodeTabWidthLowerRangeReply := #VisionDataConvert.cathodeTabWidthLowerRangeReply * 0.001;
END_REGION

REGION Network 80: Cathode Tab Length_Reply [mm](1/1000)
   RUNG wire#powerrail
      { S7_Templates := "[SrcType := DInt, DestType := Real]" } Convert(in := #VisionData.profinetInput.resultData248Byte_2[45], out => #VisionDataConvert.cathodeTabLengthReply)
      Mul(in1 := #VisionDataConvert.cathodeTabLengthReply, in2 := 0.001, out => #VisionDataConvert.cathodeTabLengthReply)
   END_RUNG
   // the same network as SCL:
   #VisionDataConvert.cathodeTabLengthReply := DINT_TO_REAL(#VisionData.profinetInput.resultData248Byte_2[45]);
   #VisionDataConvert.cathodeTabLengthReply := #VisionDataConvert.cathodeTabLengthReply * 0.001;
END_REGION

REGION Network 81: Cathode Tab Length_Upper Range Reply [mm](1/1000)
   RUNG wire#powerrail
      { S7_Templates := "[SrcType := DInt, DestType := Real]" } Convert(in := #VisionData.profinetInput.resultData248Byte_2[46], out => #VisionDataConvert.cathodeTabLengthUpperRangeReply)
      Mul(in1 := #VisionDataConvert.cathodeTabLengthUpperRangeReply, in2 := 0.001, out => #VisionDataConvert.cathodeTabLengthUpperRangeReply)
   END_RUNG
   // the same network as SCL:
   #VisionDataConvert.cathodeTabLengthUpperRangeReply := DINT_TO_REAL(#VisionData.profinetInput.resultData248Byte_2[46]);
   #VisionDataConvert.cathodeTabLengthUpperRangeReply := #VisionDataConvert.cathodeTabLengthUpperRangeReply * 0.001;
END_REGION

REGION Network 82: Cathode Tab Length_Lower Range Reply [mm](1/1000)
   RUNG wire#powerrail
      { S7_Templates := "[SrcType := DInt, DestType := Real]" } Convert(in := #VisionData.profinetInput.resultData248Byte_2[47], out => #VisionDataConvert.cathodeTabLengthLowerRangeReply)
      Mul(in1 := #VisionDataConvert.cathodeTabLengthLowerRangeReply, in2 := 0.001, out => #VisionDataConvert.cathodeTabLengthLowerRangeReply)
   END_RUNG
   // the same network as SCL:
   #VisionDataConvert.cathodeTabLengthLowerRangeReply := DINT_TO_REAL(#VisionData.profinetInput.resultData248Byte_2[47]);
   #VisionDataConvert.cathodeTabLengthLowerRangeReply := #VisionDataConvert.cathodeTabLengthLowerRangeReply * 0.001;
END_REGION

REGION Network 83: Anode Tab Width_Reply [mm](1/1000)
   RUNG wire#powerrail
      { S7_Templates := "[SrcType := DInt, DestType := Real]" } Convert(in := #VisionData.profinetInput.resultData248Byte_2[48], out => #VisionDataConvert.anodeTabWidthReply)
      Mul(in1 := #VisionDataConvert.anodeTabWidthReply, in2 := 0.001, out => #VisionDataConvert.anodeTabWidthReply)
   END_RUNG
   // the same network as SCL:
   #VisionDataConvert.anodeTabWidthReply := DINT_TO_REAL(#VisionData.profinetInput.resultData248Byte_2[48]);
   #VisionDataConvert.anodeTabWidthReply := #VisionDataConvert.anodeTabWidthReply * 0.001;
END_REGION

REGION Network 84: Anode Tab Width_Upper Range Reply [mm](1/1000)
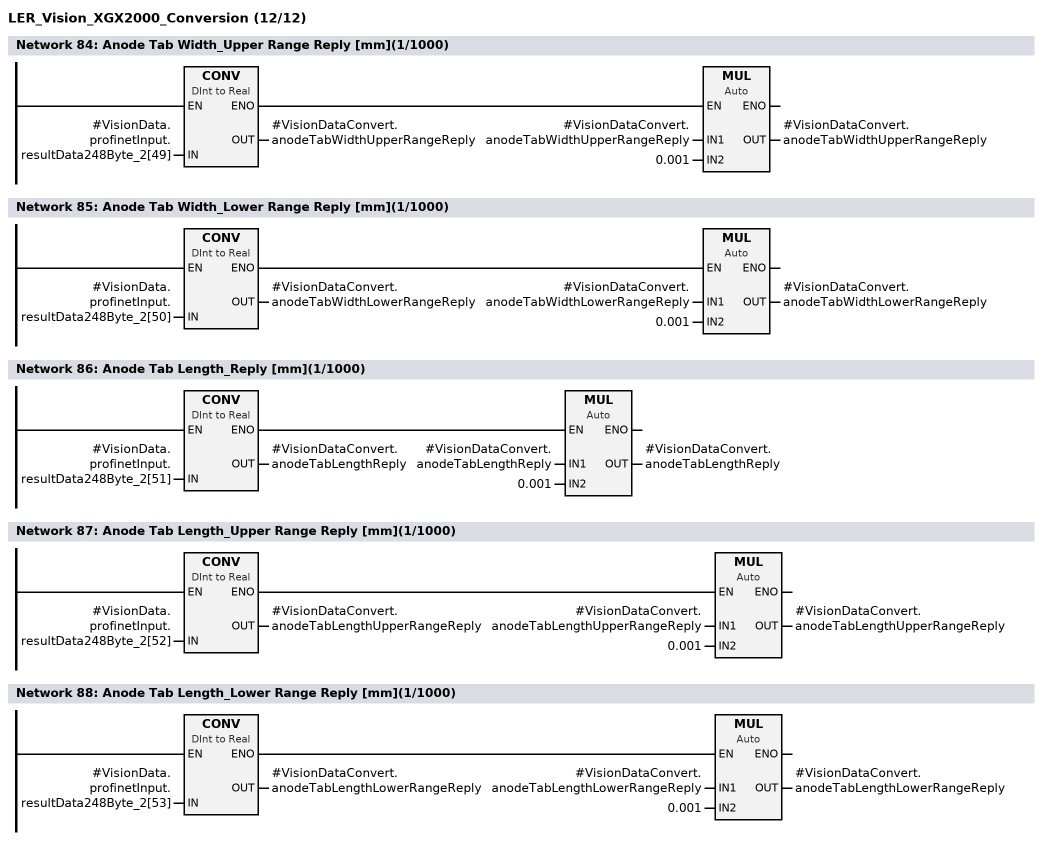
   RUNG wire#powerrail
      { S7_Templates := "[SrcType := DInt, DestType := Real]" } Convert(in := #VisionData.profinetInput.resultData248Byte_2[49], out => #VisionDataConvert.anodeTabWidthUpperRangeReply)
      Mul(in1 := #VisionDataConvert.anodeTabWidthUpperRangeReply, in2 := 0.001, out => #VisionDataConvert.anodeTabWidthUpperRangeReply)
   END_RUNG
   // the same network as SCL:
   #VisionDataConvert.anodeTabWidthUpperRangeReply := DINT_TO_REAL(#VisionData.profinetInput.resultData248Byte_2[49]);
   #VisionDataConvert.anodeTabWidthUpperRangeReply := #VisionDataConvert.anodeTabWidthUpperRangeReply * 0.001;
END_REGION

REGION Network 85: Anode Tab Width_Lower Range Reply [mm](1/1000)
   RUNG wire#powerrail
      { S7_Templates := "[SrcType := DInt, DestType := Real]" } Convert(in := #VisionData.profinetInput.resultData248Byte_2[50], out => #VisionDataConvert.anodeTabWidthLowerRangeReply)
      Mul(in1 := #VisionDataConvert.anodeTabWidthLowerRangeReply, in2 := 0.001, out => #VisionDataConvert.anodeTabWidthLowerRangeReply)
   END_RUNG
   // the same network as SCL:
   #VisionDataConvert.anodeTabWidthLowerRangeReply := DINT_TO_REAL(#VisionData.profinetInput.resultData248Byte_2[50]);
   #VisionDataConvert.anodeTabWidthLowerRangeReply := #VisionDataConvert.anodeTabWidthLowerRangeReply * 0.001;
END_REGION

REGION Network 86: Anode Tab Length_Reply [mm](1/1000)
   RUNG wire#powerrail
      { S7_Templates := "[SrcType := DInt, DestType := Real]" } Convert(in := #VisionData.profinetInput.resultData248Byte_2[51], out => #VisionDataConvert.anodeTabLengthReply)
      Mul(in1 := #VisionDataConvert.anodeTabLengthReply, in2 := 0.001, out => #VisionDataConvert.anodeTabLengthReply)
   END_RUNG
   // the same network as SCL:
   #VisionDataConvert.anodeTabLengthReply := DINT_TO_REAL(#VisionData.profinetInput.resultData248Byte_2[51]);
   #VisionDataConvert.anodeTabLengthReply := #VisionDataConvert.anodeTabLengthReply * 0.001;
END_REGION

REGION Network 87: Anode Tab Length_Upper Range Reply [mm](1/1000)
   RUNG wire#powerrail
      { S7_Templates := "[SrcType := DInt, DestType := Real]" } Convert(in := #VisionData.profinetInput.resultData248Byte_2[52], out => #VisionDataConvert.anodeTabLengthUpperRangeReply)
      Mul(in1 := #VisionDataConvert.anodeTabLengthUpperRangeReply, in2 := 0.001, out => #VisionDataConvert.anodeTabLengthUpperRangeReply)
   END_RUNG
   // the same network as SCL:
   #VisionDataConvert.anodeTabLengthUpperRangeReply := DINT_TO_REAL(#VisionData.profinetInput.resultData248Byte_2[52]);
   #VisionDataConvert.anodeTabLengthUpperRangeReply := #VisionDataConvert.anodeTabLengthUpperRangeReply * 0.001;
END_REGION

REGION Network 88: Anode Tab Length_Lower Range Reply [mm](1/1000)
   RUNG wire#powerrail
      { S7_Templates := "[SrcType := DInt, DestType := Real]" } Convert(in := #VisionData.profinetInput.resultData248Byte_2[53], out => #VisionDataConvert.anodeTabLengthLowerRangeReply)
      Mul(in1 := #VisionDataConvert.anodeTabLengthLowerRangeReply, in2 := 0.001, out => #VisionDataConvert.anodeTabLengthLowerRangeReply)
   END_RUNG
   // the same network as SCL:
   #VisionDataConvert.anodeTabLengthLowerRangeReply := DINT_TO_REAL(#VisionData.profinetInput.resultData248Byte_2[53]);
   #VisionDataConvert.anodeTabLengthLowerRangeReply := #VisionDataConvert.anodeTabLengthLowerRangeReply * 0.001;
END_REGION
END_FUNCTION_BLOCK
